LIN {X 0,Y 305.472,Z 165.433,A -85,B 0,C 180,E1 -15814.078,E2 -15814.078} C_VEL
LIN {X 0,Y 305.453,Z 165.439,A -85,B 0,C 180,E1 -15818.399,E2 -15818.399} C_VEL
LIN {X 0,Y 305.502,Z 165.428,A -85,B 0,C 180,E1 -15821.212,E2 -15821.212} C_VEL
LIN {X 0,Y 305.572,Z 165.418,A -85,B 0,C 180,E1 -15825.345,E2 -15825.345} C_VEL
LIN {X 0,Y 305.615,Z 165.414,A -85,B 0,C 180,E1 -15829.399,E2 -15829.399} C_VEL
LIN {X 0,Y 305.74,Z 165.403,A -85,B 0,C 180,E1 -15832.072,E2 -15832.072} C_VEL
LIN {X 0,Y 305.65,Z 165.409,A -85,B 0,C 180,E1 -15834.722,E2 -15834.722} C_VEL
LIN {X 0,Y 305.927,Z 165.375,A -85,B 0,C 180,E1 -15838.683,E2 -15838.683} C_VEL
LIN {X 0,Y 305.927,Z 165.375,A -85,B 0,C 180,E1 -15841.316,E2 -15841.316} C_VEL
LIN {X 0,Y 305.778,Z 165.393,A -85,B 0,C 180,E1 -15846.599,E2 -15846.599} C_VEL
LIN {X 0,Y 305.687,Z 165.406,A -85,B 0,C 180,E1 -15849.261,E2 -15849.261} C_VEL
LIN {X 0,Y 305.562,Z 165.422,A -85,B 0,C 180,E1 -15853.297,E2 -15853.297} C_VEL
LIN {X 0,Y 305.503,Z 165.429,A -85,B 0,C 180,E1 -15856.025,E2 -15856.025} C_VEL
LIN {X 0,Y 305.465,Z 165.432,A -85,B 0,C 180,E1 -15860.189,E2 -15860.189} C_VEL
LIN {X 0,Y 305.432,Z 165.436,A -85,B 0,C 180,E1 -15864.468,E2 -15864.468} C_VEL
LIN {X 0,Y 305.441,Z 165.44,A -85,B 0,C 180,E1 -15867.399,E2 -15867.399} C_VEL
LIN {X 0,Y 305.422,Z 165.437,A -85,B 0,C 180,E1 -15870.413,E2 -15870.413} C_VEL
LIN {X 0,Y 305.458,Z 165.433,A -85,B 0,C 180,E1 -15874.079,E2 -15874.079} C_VEL
LIN {X 0,Y 305.446,Z 165.435,A -85,B 0,C 180,E1 -15876.743,E2 -15876.743} C_VEL
LIN {X 0,Y 305.403,Z 165.441,A -85,B 0,C 180,E1 -15880.59,E2 -15880.59} C_VEL
LIN {X 0,Y 305.414,Z 165.439,A -85,B 0,C 180,E1 -15883.657,E2 -15883.657} C_VEL
LIN {X 0,Y 305.429,Z 165.438,A -85,B 0,C 180,E1 -15887.42,E2 -15887.42} C_VEL
LIN {X 0,Y 305.455,Z 165.434,A -85,B 0,C 180,E1 -15891.596,E2 -15891.596} C_VEL
LIN {X 0,Y 305.457,Z 165.438,A -85,B 0,C 180,E1 -15894.888,E2 -15894.888} C_VEL
LIN {X 0,Y 305.476,Z 165.491,A -85,B 0,C 180,E1 -15898.875,E2 -15898.875} C_VEL
LIN {X 0,Y 308.066,Z 178.627,A -85,B 0,C 180,E1 -15902.855,E2 -15902.855} C_VEL
LIN {X 0,Y 309.134,Z 185.066,A -85,B 0,C 180,E1 -15904.733,E2 -15904.733} C_VEL
LIN {X 0,Y 308.784,Z 188.883,A -85,B 0,C 180,E1 -15905.779,E2 -15905.779} C_VEL
LIN {X 0,Y 313.815,Z 227.795,A -85,B 0,C 180,E1 -15907.228,E2 -15907.228} C_VEL
LIN {X 0,Y 311.768,Z 298.034,A -85,B 0,C 180,E1 -15909.205,E2 -15909.205} C_VEL
LIN {X 0,Y 311.014,Z 311.572,A -85,B 0,C 180,E1 -15909.844,E2 -15909.844} C_VEL
LIN {X 0,Y 310.145,Z 323.511,A -85,B 0,C 180,E1 -15910.647,E2 -15910.647} C_VEL
LIN {X 0,Y 309.009,Z 336.037,A -85,B 0,C 180,E1 -15911.778,E2 -15911.778} C_VEL
LIN {X 0,Y 307.83,Z 347.584,A -85,B 0,C 180,E1 -15913.112,E2 -15913.112} C_VEL
LIN {X 0,Y 306.764,Z 358.549,A -85,B 0,C 180,E1 -15914.725,E2 -15914.725} C_VEL
LIN {X 0,Y 305.802,Z 367.631,A -85,B 0,C 180,E1 -15916.376,E2 -15916.376} C_VEL
LIN {X 0,Y 304.946,Z 375.108,A -85,B 0,C 180,E1 -15918.03,E2 -15918.03} C_VEL
LIN {X 0,Y 304.346,Z 382.452,A -85,B 0,C 180,E1 -15920.028,E2 -15920.028} C_VEL
LIN {X 0,Y 303.939,Z 388.258,A -85,B 0,C 180,E1 -15922.026,E2 -15922.026} C_VEL
LIN {X 0,Y 303.666,Z 393.461,A -85,B 0,C 180,E1 -15924.375,E2 -15924.375} C_VEL
LIN {X 0,Y 303.654,Z 396.168,A -85,B 0,C 180,E1 -15926.02,E2 -15926.02} C_VEL
LIN {X 0,Y 303.618,Z 397.825,A -85,B 0,C 180,E1 -15927.348,E2 -15927.348} C_VEL
LIN {X 0,Y 303.582,Z 399.055,A -85,B 0,C 180,E1 -15928.675,E2 -15928.675} C_VEL
LIN {X 0,Y 303.607,Z 399.819,A -85,B 0,C 180,E1 -15930.001,E2 -15930.001} C_VEL
LIN {X 0,Y 303.565,Z 400.151,A -85,B 0,C 180,E1 -15931.328,E2 -15931.328} C_VEL
LIN {X 0,Y 303.601,Z 400.076,A -85,B 0,C 180,E1 -15932.655,E2 -15932.655} C_VEL
LIN {X 0,Y 303.591,Z 399.592,A -85,B 0,C 180,E1 -15933.983,E2 -15933.983} C_VEL
LIN {X 0,Y 303.625,Z 398.44,A -85,B 0,C 180,E1 -15935.546,E2 -15935.546} C_VEL
LIN {X 0,Y 304.036,Z 395.535,A -85,B 0,C 180,E1 -15937.973,E2 -15937.973} C_VEL
LIN {X 0,Y 304.61,Z 392.021,A -85,B 0,C 180,E1 -15939.966,E2 -15939.966} C_VEL
LIN {X 0,Y 305.477,Z 387.416,A -85,B 0,C 180,E1 -15941.951,E2 -15941.951} C_VEL
LIN {X 0,Y 306.627,Z 381.601,A -85,B 0,C 180,E1 -15943.927,E2 -15943.927} C_VEL
LIN {X 0,Y 308.262,Z 374.337,A -85,B 0,C 180,E1 -15945.879,E2 -15945.879} C_VEL
LIN {X 0,Y 310.051,Z 365.064,A -85,B 0,C 180,E1 -15947.882,E2 -15947.882} C_VEL
LIN {X 0,Y 312.002,Z 355.271,A -85,B 0,C 180,E1 -15949.578,E2 -15949.578} C_VEL
LIN {X 0,Y 314.276,Z 343.752,A -85,B 0,C 180,E1 -15951.138,E2 -15951.138} C_VEL
LIN {X 0,Y 316.217,Z 332.295,A -85,B 0,C 180,E1 -15952.372,E2 -15952.372} C_VEL
LIN {X 0,Y 317.969,Z 319.356,A -85,B 0,C 180,E1 -15953.445,E2 -15953.445} C_VEL
LIN {X 0,Y 319.623,Z 306.314,A -85,B 0,C 180,E1 -15954.22,E2 -15954.22} C_VEL
LIN {X 0,Y 320.675,Z 292.777,A -85,B 0,C 180,E1 -15954.774,E2 -15954.774} C_VEL
LIN {X 0,Y 323.701,Z 230.457,A -85,B 0,C 180,E1 -15956.607,E2 -15956.607} C_VEL
LIN {X 0,Y 321.649,Z 216.499,A -85,B 0,C 180,E1 -15957.392,E2 -15957.392} C_VEL
LIN {X 0,Y 318.885,Z 202.613,A -85,B 0,C 180,E1 -15958.296,E2 -15958.296} C_VEL
LIN {X 0,Y 314.226,Z 192.61,A -85,B 0,C 180,E1 -15959.393,E2 -15959.393} C_VEL
LIN {X 0,Y 311.037,Z 185.839,A -85,B 0,C 180,E1 -15960.213,E2 -15960.213} C_VEL
LIN {X 0,Y 309.147,Z 178.305,A -85,B 0,C 180,E1 -15963.067,E2 -15963.067} C_VEL
LIN {X 0,Y 307.457,Z 172.034,A -85,B 0,C 180,E1 -15965.654,E2 -15965.654} C_VEL
LIN {X 0,Y 305.463,Z 165.437,A -85,B 0,C 180,E1 -15968.727,E2 -15968.727} C_VEL
LIN {X 0,Y 305.437,Z 165.436,A -85,B 0,C 180,E1 -15972.582,E2 -15972.582} C_VEL
LIN {X 0,Y 305.424,Z 165.43,A -85,B 0,C 180,E1 -15976.345,E2 -15976.345} C_VEL
LIN {X 0,Y 305.413,Z 165.437,A -85,B 0,C 180,E1 -15979.885,E2 -15979.885} C_VEL
LIN {X 0,Y 305.465,Z 165.429,A -85,B 0,C 180,E1 -15983.637,E2 -15983.637} C_VEL
LIN {X 0,Y 305.468,Z 165.43,A -85,B 0,C 180,E1 -15986.484,E2 -15986.484} C_VEL
LIN {X 0,Y 305.433,Z 165.434,A -85,B 0,C 180,E1 -15989.588,E2 -15989.588} C_VEL
LIN {X 0,Y 305.453,Z 165.433,A -85,B 0,C 180,E1 -15992.602,E2 -15992.602} C_VEL
LIN {X 0,Y 305.459,Z 165.434,A -85,B 0,C 180,E1 -15995.535,E2 -15995.535} C_VEL
LIN {X 0,Y 305.483,Z 165.428,A -85,B 0,C 180,E1 -15999.813,E2 -15999.813} C_VEL
LIN {X 0,Y 305.518,Z 165.426,A -85,B 0,C 180,E1 -16003.976,E2 -16003.976} C_VEL
LIN {X 0,Y 305.576,Z 165.421,A -85,B 0,C 180,E1 -16006.704,E2 -16006.704} C_VEL
LIN {X 0,Y 305.758,Z 165.403,A -85,B 0,C 180,E1 -16011.262,E2 -16011.262} C_VEL
LIN {X 0,Y 305.814,Z 165.503,A -85,B 0,C 180,E1 -16013.319,E2 -16013.319} C_VEL
LIN {X 0,Y 308.783,Z 174.874,A -85,B 0,C 180,E1 -16017.493,E2 -16017.493} C_VEL
LIN {X 0,Y 316.098,Z 187.842,A -85,B 0,C 180,E1 -16019.227,E2 -16019.227} C_VEL
LIN {X 0,Y 320.795,Z 197.781,A -85,B 0,C 180,E1 -16020.318,E2 -16020.318} C_VEL
LIN {X 0,Y 324.339,Z 206.07,A -85,B 0,C 180,E1 -16021.105,E2 -16021.105} C_VEL
LIN {X 0,Y 324.803,Z 209.109,A -85,B 0,C 180,E1 -16021.277,E2 -16021.277} C_VEL
LIN {X 0,Y 320.791,Z 283.034,A -85,B 0,C 180,E1 -16023.454,E2 -16023.454} C_VEL
LIN {X 0,Y 319.653,Z 296.49,A -85,B 0,C 180,E1 -16024.098,E2 -16024.098} C_VEL
LIN {X 0,Y 318.359,Z 308.395,A -85,B 0,C 180,E1 -16024.908,E2 -16024.908} C_VEL
LIN {X 0,Y 316.679,Z 320.8,A -85,B 0,C 180,E1 -16026.033,E2 -16026.033} C_VEL
LIN {X 0,Y 314.754,Z 332.399,A -85,B 0,C 180,E1 -16027.377,E2 -16027.377} C_VEL
LIN {X 0,Y 312.921,Z 342.14,A -85,B 0,C 180,E1 -16028.802,E2 -16028.802} C_VEL
LIN {X 0,Y 311.039,Z 351.123,A -85,B 0,C 180,E1 -16030.415,E2 -16030.415} C_VEL
LIN {X 0,Y 309.272,Z 359.452,A -85,B 0,C 180,E1 -16032.269,E2 -16032.269} C_VEL
LIN {X 0,Y 307.722,Z 366.472,A -85,B 0,C 180,E1 -16034.213,E2 -16034.213} C_VEL
LIN {X 0,Y 306.509,Z 371.582,A -85,B 0,C 180,E1 -16035.971,E2 -16035.971} C_VEL
LIN {X 0,Y 305.397,Z 376.396,A -85,B 0,C 180,E1 -16038.1,E2 -16038.1} C_VEL
LIN {X 0,Y 304.623,Z 379.954,A -85,B 0,C 180,E1 -16040.247,E2 -16040.247} C_VEL
LIN {X 0,Y 304.009,Z 382.327,A -85,B 0,C 180,E1 -16042.373,E2 -16042.373} C_VEL
LIN {X 0,Y 303.584,Z 383.655,A -85,B 0,C 180,E1 -16044.627,E2 -16044.627} C_VEL
LIN {X 0,Y 303.405,Z 383.901,A -85,B 0,C 180,E1 -16046.112,E2 -16046.112} C_VEL
LIN {X 0,Y 303.329,Z 383.27,A -85,B 0,C 180,E1 -16048.302,E2 -16048.302} C_VEL
LIN {X 0,Y 303.429,Z 380.868,A -85,B 0,C 180,E1 -16051.018,E2 -16051.018} C_VEL
LIN {X 0,Y 303.701,Z 378.144,A -85,B 0,C 180,E1 -16052.891,E2 -16052.891} C_VEL
LIN {X 0,Y 304.053,Z 373.262,A -85,B 0,C 180,E1 -16055.301,E2 -16055.301} C_VEL
LIN {X 0,Y 304.626,Z 366.761,A -85,B 0,C 180,E1 -16057.64,E2 -16057.64} C_VEL
LIN {X 0,Y 305.372,Z 359.46,A -85,B 0,C 180,E1 -16059.692,E2 -16059.692} C_VEL
LIN {X 0,Y 306.156,Z 351.81,A -85,B 0,C 180,E1 -16061.427,E2 -16061.427} C_VEL
LIN {X 0,Y 307.049,Z 342.979,A -85,B 0,C 180,E1 -16063.065,E2 -16063.065} C_VEL
LIN {X 0,Y 308.206,Z 331.704,A -85,B 0,C 180,E1 -16064.753,E2 -16064.753} C_VEL
LIN {X 0,Y 309.372,Z 319.69,A -85,B 0,C 180,E1 -16066.164,E2 -16066.164} C_VEL
LIN {X 0,Y 310.388,Z 307.413,A -85,B 0,C 180,E1 -16067.287,E2 -16067.287} C_VEL
LIN {X 0,Y 311.251,Z 294.444,A -85,B 0,C 180,E1 -16068.172,E2 -16068.172} C_VEL
LIN {X 0,Y 311.848,Z 281.457,A -85,B 0,C 180,E1 -16068.79,E2 -16068.79} C_VEL
LIN {X 0,Y 313.435,Z 231.762,A -85,B 0,C 180,E1 -16070.193,E2 -16070.193} C_VEL
LIN {X 0,Y 314.134,Z 202.407,A -85,B 0,C 180,E1 -16071.018,E2 -16071.018} C_VEL
LIN {X 0,Y 311.365,Z 186.836,A -85,B 0,C 180,E1 -16071.635,E2 -16071.635} C_VEL
LIN {X 0,Y 306.865,Z 172.397,A -85,B 0,C 180,E1 -16072.373,E2 -16072.373} C_VEL
LIN {X 0,Y 305.523,Z 165.429,A -85,B 0,C 180,E1 -16074.692,E2 -16074.692} C_VEL
LIN {X 0,Y 305.447,Z 165.439,A -85,B 0,C 180,E1 -16078.358,E2 -16078.358} C_VEL
LIN {X 0,Y 305.458,Z 165.434,A -85,B 0,C 180,E1 -16081.106,E2 -16081.106} C_VEL
LIN {X 0,Y 305.483,Z 165.433,A -85,B 0,C 180,E1 -16084.079,E2 -16084.079} C_VEL
LIN {X 0,Y 305.463,Z 165.436,A -85,B 0,C 180,E1 -16088.399,E2 -16088.399} C_VEL
LIN {X 0,Y 305.506,Z 165.427,A -85,B 0,C 180,E1 -16091.211,E2 -16091.211} C_VEL
LIN {X 0,Y 305.583,Z 165.418,A -85,B 0,C 180,E1 -16095.345,E2 -16095.345} C_VEL
LIN {X 0,Y 305.627,Z 165.413,A -85,B 0,C 180,E1 -16099.398,E2 -16099.398} C_VEL
LIN {X 0,Y 305.751,Z 165.401,A -85,B 0,C 180,E1 -16102.072,E2 -16102.072} C_VEL
LIN {X 0,Y 305.66,Z 165.408,A -85,B 0,C 180,E1 -16104.722,E2 -16104.722} C_VEL
LIN {X 0,Y 305.939,Z 165.373,A -85,B 0,C 180,E1 -16108.683,E2 -16108.683} C_VEL
LIN {X 0,Y 305.939,Z 165.374,A -85,B 0,C 180,E1 -16111.315,E2 -16111.315} C_VEL
LIN {X 0,Y 305.787,Z 165.392,A -85,B 0,C 180,E1 -16116.598,E2 -16116.598} C_VEL
LIN {X 0,Y 305.697,Z 165.405,A -85,B 0,C 180,E1 -16119.26,E2 -16119.26} C_VEL
LIN {X 0,Y 305.572,Z 165.422,A -85,B 0,C 180,E1 -16123.296,E2 -16123.296} C_VEL
LIN {X 0,Y 305.512,Z 165.427,A -85,B 0,C 180,E1 -16126.023,E2 -16126.023} C_VEL
LIN {X 0,Y 305.473,Z 165.431,A -85,B 0,C 180,E1 -16130.187,E2 -16130.187} C_VEL
LIN {X 0,Y 305.44,Z 165.435,A -85,B 0,C 180,E1 -16134.466,E2 -16134.466} C_VEL
LIN {X 0,Y 305.449,Z 165.438,A -85,B 0,C 180,E1 -16137.397,E2 -16137.397} C_VEL
LIN {X 0,Y 305.428,Z 165.437,A -85,B 0,C 180,E1 -16140.411,E2 -16140.411} C_VEL
LIN {X 0,Y 305.463,Z 165.432,A -85,B 0,C 180,E1 -16144.077,E2 -16144.077} C_VEL
LIN {X 0,Y 305.451,Z 165.436,A -85,B 0,C 180,E1 -16146.741,E2 -16146.741} C_VEL
LIN {X 0,Y 305.407,Z 165.441,A -85,B 0,C 180,E1 -16150.588,E2 -16150.588} C_VEL
LIN {X 0,Y 305.418,Z 165.438,A -85,B 0,C 180,E1 -16153.655,E2 -16153.655} C_VEL
LIN {X 0,Y 305.431,Z 165.437,A -85,B 0,C 180,E1 -16157.417,E2 -16157.417} C_VEL
LIN {X 0,Y 305.456,Z 165.433,A -85,B 0,C 180,E1 -16161.594,E2 -16161.594} C_VEL
LIN {X 0,Y 305.441,Z 165.435,A -85,B 0,C 180,E1 -16164.445,E2 -16164.445} C_VEL
LIN {X 0,Y 304.777,Z 165.521,A -85,B 0,C 180,E1 -16165.546,E2 -16165.546} C_VEL
LIN {X 0,Y 301.877,Z 165.879,A -85,B 0,C 180,E1 -16167.337,E2 -16167.337} C_VEL
LIN {X 0,Y 299.44,Z 166.186,A -85,B 0,C 180,E1 -16168.791,E2 -16168.791} C_VEL
LIN {X 0,Y 298.44,Z 166.308,A -85,B 0,C 180,E1 -16169.918,E2 -16169.918} C_VEL
LIN {X 0,Y 298.383,Z 166.317,A -85,B 0,C 180,E1 -16170.299,E2 -16170.299} C_VEL
LIN {X 0,Y 298.398,Z 166.312,A -85,B 0,C 180,E1 -16173.504,E2 -16173.504} C_VEL
LIN {X 0,Y 298.399,Z 166.314,A -85,B 0,C 180,E1 -16176.71,E2 -16176.71} C_VEL
LIN {X 0,Y 298.453,Z 166.307,A -85,B 0,C 180,E1 -16180.751,E2 -16180.751} C_VEL
LIN {X 0,Y 298.504,Z 166.299,A -85,B 0,C 180,E1 -16184.99,E2 -16184.99} C_VEL
LIN {X 0,Y 298.574,Z 166.291,A -85,B 0,C 180,E1 -16189.146,E2 -16189.146} C_VEL
LIN {X 0,Y 298.691,Z 166.279,A -85,B 0,C 180,E1 -16191.884,E2 -16191.884} C_VEL
LIN {X 0,Y 298.62,Z 166.285,A -85,B 0,C 180,E1 -16194.598,E2 -16194.598} C_VEL
LIN {X 0,Y 298.895,Z 166.251,A -85,B 0,C 180,E1 -16198.652,E2 -16198.652} C_VEL
LIN {X 0,Y 298.895,Z 166.251,A -85,B 0,C 180,E1 -16201.347,E2 -16201.347} C_VEL
LIN {X 0,Y 298.727,Z 166.271,A -85,B 0,C 180,E1 -16206.755,E2 -16206.755} C_VEL
LIN {X 0,Y 298.618,Z 166.288,A -85,B 0,C 180,E1 -16209.482,E2 -16209.482} C_VEL
LIN {X 0,Y 298.515,Z 166.303,A -85,B 0,C 180,E1 -16213.617,E2 -16213.617} C_VEL
LIN {X 0,Y 298.443,Z 166.307,A -85,B 0,C 180,E1 -16216.414,E2 -16216.414} C_VEL
LIN {X 0,Y 298.422,Z 166.314,A -85,B 0,C 180,E1 -16219.61,E2 -16219.61} C_VEL
LIN {X 0,Y 298.375,Z 166.319,A -85,B 0,C 180,E1 -16223.604,E2 -16223.604} C_VEL
LIN {X 0,Y 298.395,Z 166.313,A -85,B 0,C 180,E1 -16226.583,E2 -16226.583} C_VEL
LIN {X 0,Y 298.385,Z 166.316,A -85,B 0,C 180,E1 -16229.645,E2 -16229.645} C_VEL
LIN {X 0,Y 298.386,Z 166.315,A -85,B 0,C 180,E1 -16232.801,E2 -16232.801} C_VEL
LIN {X 0,Y 298.421,Z 166.311,A -85,B 0,C 180,E1 -16236.803,E2 -16236.803} C_VEL
LIN {X 0,Y 298.367,Z 166.318,A -85,B 0,C 180,E1 -16239.493,E2 -16239.493} C_VEL
LIN {X 0,Y 298.364,Z 166.322,A -85,B 0,C 180,E1 -16243.098,E2 -16243.098} C_VEL
LIN {X 0,Y 298.365,Z 166.322,A -85,B 0,C 180,E1 -16246.916,E2 -16246.916} C_VEL
LIN {X 0,Y 298.379,Z 166.319,A -85,B 0,C 180,E1 -16251.012,E2 -16251.012} C_VEL
LIN {X 0,Y 298.4,Z 166.312,A -85,B 0,C 180,E1 -16253.929,E2 -16253.929} C_VEL
LIN {X 0,Y 298.389,Z 166.317,A -85,B 0,C 180,E1 -16257.201,E2 -16257.201} C_VEL
LIN {X 0,Y 298.415,Z 166.357,A -85,B 0,C 180,E1 -16258.581,E2 -16258.581} C_VEL
LIN {X 0,Y 300.976,Z 179.093,A -85,B 0,C 180,E1 -16262.539,E2 -16262.539} C_VEL
LIN {X 0,Y 302.103,Z 185.693,A -85,B 0,C 180,E1 -16264.511,E2 -16264.511} C_VEL
LIN {X 0,Y 301.911,Z 188.736,A -85,B 0,C 180,E1 -16265.371,E2 -16265.371} C_VEL
LIN {X 0,Y 306.968,Z 229.189,A -85,B 0,C 180,E1 -16266.912,E2 -16266.912} C_VEL
LIN {X 0,Y 304.887,Z 297.637,A -85,B 0,C 180,E1 -16268.89,E2 -16268.89} C_VEL
LIN {X 0,Y 304.135,Z 311.222,A -85,B 0,C 180,E1 -16269.544,E2 -16269.544} C_VEL
LIN {X 0,Y 303.23,Z 323.192,A -85,B 0,C 180,E1 -16270.364,E2 -16270.364} C_VEL
LIN {X 0,Y 302.05,Z 335.742,A -85,B 0,C 180,E1 -16271.518,E2 -16271.518} C_VEL
LIN {X 0,Y 300.83,Z 347.439,A -85,B 0,C 180,E1 -16272.9,E2 -16272.9} C_VEL
LIN {X 0,Y 299.791,Z 357.614,A -85,B 0,C 180,E1 -16274.417,E2 -16274.417} C_VEL
LIN {X 0,Y 298.817,Z 366.553,A -85,B 0,C 180,E1 -16276.051,E2 -16276.051} C_VEL
LIN {X 0,Y 297.828,Z 375.581,A -85,B 0,C 180,E1 -16278.085,E2 -16278.085} C_VEL
LIN {X 0,Y 297.207,Z 382.758,A -85,B 0,C 180,E1 -16280.13,E2 -16280.13} C_VEL
LIN {X 0,Y 296.785,Z 389.304,A -85,B 0,C 180,E1 -16282.518,E2 -16282.518} C_VEL
LIN {X 0,Y 296.58,Z 393.545,A -85,B 0,C 180,E1 -16284.562,E2 -16284.562} C_VEL
LIN {X 0,Y 296.566,Z 395.739,A -85,B 0,C 180,E1 -16285.924,E2 -16285.924} C_VEL
LIN {X 0,Y 296.545,Z 397.441,A -85,B 0,C 180,E1 -16287.284,E2 -16287.284} C_VEL
LIN {X 0,Y 296.501,Z 398.713,A -85,B 0,C 180,E1 -16288.643,E2 -16288.643} C_VEL
LIN {X 0,Y 296.521,Z 399.555,A -85,B 0,C 180,E1 -16290.001,E2 -16290.001} C_VEL
LIN {X 0,Y 296.485,Z 399.929,A -85,B 0,C 180,E1 -16291.359,E2 -16291.359} C_VEL
LIN {X 0,Y 296.525,Z 399.894,A -85,B 0,C 180,E1 -16292.718,E2 -16292.718} C_VEL
LIN {X 0,Y 296.491,Z 399.454,A -85,B 0,C 180,E1 -16294.079,E2 -16294.079} C_VEL
LIN {X 0,Y 296.546,Z 398.537,A -85,B 0,C 180,E1 -16295.51,E2 -16295.51} C_VEL
LIN {X 0,Y 296.986,Z 395.571,A -85,B 0,C 180,E1 -16298.164,E2 -16298.164} C_VEL
LIN {X 0,Y 297.591,Z 392.145,A -85,B 0,C 180,E1 -16300.203,E2 -16300.203} C_VEL
LIN {X 0,Y 298.507,Z 387.63,A -85,B 0,C 180,E1 -16302.235,E2 -16302.235} C_VEL
LIN {X 0,Y 299.758,Z 381.92,A -85,B 0,C 180,E1 -16304.253,E2 -16304.253} C_VEL
LIN {X 0,Y 301.466,Z 374.857,A -85,B 0,C 180,E1 -16306.247,E2 -16306.247} C_VEL
LIN {X 0,Y 303.31,Z 365.962,A -85,B 0,C 180,E1 -16308.257,E2 -16308.257} C_VEL
LIN {X 0,Y 305.241,Z 357.152,A -85,B 0,C 180,E1 -16309.854,E2 -16309.854} C_VEL
LIN {X 0,Y 307.472,Z 346.24,A -85,B 0,C 180,E1 -16311.453,E2 -16311.453} C_VEL
LIN {X 0,Y 309.771,Z 333.801,A -85,B 0,C 180,E1 -16312.864,E2 -16312.864} C_VEL
LIN {X 0,Y 311.583,Z 321.633,A -85,B 0,C 180,E1 -16313.955,E2 -16313.955} C_VEL
LIN {X 0,Y 313.417,Z 308.119,A -85,B 0,C 180,E1 -16314.82,E2 -16314.82} C_VEL
LIN {X 0,Y 314.688,Z 294.787,A -85,B 0,C 180,E1 -16315.419,E2 -16315.419} C_VEL
LIN {X 0,Y 317.963,Z 231.766,A -85,B 0,C 180,E1 -16317.319,E2 -16317.319} C_VEL
LIN {X 0,Y 315.972,Z 217.769,A -85,B 0,C 180,E1 -16318.133,E2 -16318.133} C_VEL
LIN {X 0,Y 313.691,Z 206.025,A -85,B 0,C 180,E1 -16318.94,E2 -16318.94} C_VEL
LIN {X 0,Y 308.299,Z 194.321,A -85,B 0,C 180,E1 -16320.281,E2 -16320.281} C_VEL
LIN {X 0,Y 305.45,Z 188.925,A -85,B 0,C 180,E1 -16321.007,E2 -16321.007} C_VEL
LIN {X 0,Y 303.831,Z 185.519,A -85,B 0,C 180,E1 -16321.484,E2 -16321.484} C_VEL
LIN {X 0,Y 301.449,Z 176.169,A -85,B 0,C 180,E1 -16325.314,E2 -16325.314} C_VEL
LIN {X 0,Y 299.296,Z 169.326,A -85,B 0,C 180,E1 -16328.55,E2 -16328.55} C_VEL
LIN {X 0,Y 298.379,Z 166.317,A -85,B 0,C 180,E1 -16330.151,E2 -16330.151} C_VEL
LIN {X 0,Y 298.373,Z 166.315,A -85,B 0,C 180,E1 -16333.098,E2 -16333.098} C_VEL
LIN {X 0,Y 298.373,Z 166.309,A -85,B 0,C 180,E1 -16336.916,E2 -16336.916} C_VEL
LIN {X 0,Y 298.388,Z 166.308,A -85,B 0,C 180,E1 -16341.012,E2 -16341.012} C_VEL
LIN {X 0,Y 298.407,Z 166.308,A -85,B 0,C 180,E1 -16343.929,E2 -16343.929} C_VEL
LIN {X 0,Y 298.396,Z 166.313,A -85,B 0,C 180,E1 -16347.2,E2 -16347.2} C_VEL
LIN {X 0,Y 298.405,Z 166.314,A -85,B 0,C 180,E1 -16350.626,E2 -16350.626} C_VEL
LIN {X 0,Y 298.425,Z 166.307,A -85,B 0,C 180,E1 -16354.919,E2 -16354.919} C_VEL
LIN {X 0,Y 298.419,Z 166.306,A -85,B 0,C 180,E1 -16359.313,E2 -16359.313} C_VEL
LIN {X 0,Y 298.452,Z 166.306,A -85,B 0,C 180,E1 -16362.174,E2 -16362.174} C_VEL
LIN {X 0,Y 298.515,Z 166.303,A -85,B 0,C 180,E1 -16364.991,E2 -16364.991} C_VEL
LIN {X 0,Y 298.587,Z 166.296,A -85,B 0,C 180,E1 -16369.147,E2 -16369.147} C_VEL
LIN {X 0,Y 298.713,Z 166.37,A -85,B 0,C 180,E1 -16371.885,E2 -16371.885} C_VEL
LIN {X 0,Y 299.956,Z 170.371,A -85,B 0,C 180,E1 -16373.948,E2 -16373.948} C_VEL
LIN {X 0,Y 301.337,Z 175.242,A -85,B 0,C 180,E1 -16376.139,E2 -16376.139} C_VEL
LIN {X 0,Y 304.291,Z 179.547,A -85,B 0,C 180,E1 -16376.897,E2 -16376.897} C_VEL
LIN {X 0,Y 311.305,Z 192.016,A -85,B 0,C 180,E1 -16378.646,E2 -16378.646} C_VEL
LIN {X 0,Y 316.01,Z 202.117,A -85,B 0,C 180,E1 -16379.779,E2 -16379.779} C_VEL
LIN {X 0,Y 318.965,Z 209.24,A -85,B 0,C 180,E1 -16380.494,E2 -16380.494} C_VEL
LIN {X 0,Y 318.072,Z 227.571,A -85,B 0,C 180,E1 -16381.061,E2 -16381.061} C_VEL
LIN {X 0,Y 314.991,Z 282.686,A -85,B 0,C 180,E1 -16382.718,E2 -16382.718} C_VEL
LIN {X 0,Y 313.782,Z 296.248,A -85,B 0,C 180,E1 -16383.371,E2 -16383.371} C_VEL
LIN {X 0,Y 312.23,Z 309.274,A -85,B 0,C 180,E1 -16384.276,E2 -16384.276} C_VEL
LIN {X 0,Y 310.419,Z 321.832,A -85,B 0,C 180,E1 -16385.46,E2 -16385.46} C_VEL
LIN {X 0,Y 308.303,Z 333.575,A -85,B 0,C 180,E1 -16386.874,E2 -16386.874} C_VEL
LIN {X 0,Y 306.059,Z 344.76,A -85,B 0,C 180,E1 -16388.592,E2 -16388.592} C_VEL
LIN {X 0,Y 304.069,Z 353.697,A -85,B 0,C 180,E1 -16390.319,E2 -16390.319} C_VEL
LIN {X 0,Y 302.142,Z 361.956,A -85,B 0,C 180,E1 -16392.323,E2 -16392.323} C_VEL
LIN {X 0,Y 300.35,Z 369.263,A -85,B 0,C 180,E1 -16394.569,E2 -16394.569} C_VEL
LIN {X 0,Y 298.812,Z 375.42,A -85,B 0,C 180,E1 -16397.098,E2 -16397.098} C_VEL
LIN {X 0,Y 297.873,Z 379.354,A -85,B 0,C 180,E1 -16399.305,E2 -16399.305} C_VEL
LIN {X 0,Y 297.361,Z 381.278,A -85,B 0,C 180,E1 -16400.764,E2 -16400.764} C_VEL
LIN {X 0,Y 296.879,Z 382.975,A -85,B 0,C 180,E1 -16402.592,E2 -16402.592} C_VEL
LIN {X 0,Y 296.632,Z 383.657,A -85,B 0,C 180,E1 -16403.752,E2 -16403.752} C_VEL
LIN {X 0,Y 296.374,Z 384.096,A -85,B 0,C 180,E1 -16405.694,E2 -16405.694} C_VEL
LIN {X 0,Y 296.238,Z 383.358,A -85,B 0,C 180,E1 -16408.326,E2 -16408.326} C_VEL
LIN {X 0,Y 296.262,Z 382.178,A -85,B 0,C 180,E1 -16409.879,E2 -16409.879} C_VEL
LIN {X 0,Y 296.51,Z 379.335,A -85,B 0,C 180,E1 -16412.23,E2 -16412.23} C_VEL
LIN {X 0,Y 296.872,Z 374.965,A -85,B 0,C 180,E1 -16414.623,E2 -16414.623} C_VEL
LIN {X 0,Y 297.194,Z 370.485,A -85,B 0,C 180,E1 -16416.482,E2 -16416.482} C_VEL
LIN {X 0,Y 297.764,Z 364.753,A -85,B 0,C 180,E1 -16418.384,E2 -16418.384} C_VEL
LIN {X 0,Y 298.532,Z 357.413,A -85,B 0,C 180,E1 -16420.347,E2 -16420.347} C_VEL
LIN {X 0,Y 299.483,Z 348.857,A -85,B 0,C 180,E1 -16422.202,E2 -16422.202} C_VEL
LIN {X 0,Y 300.445,Z 339.005,A -85,B 0,C 180,E1 -16423.93,E2 -16423.93} C_VEL
LIN {X 0,Y 301.689,Z 327.13,A -85,B 0,C 180,E1 -16425.586,E2 -16425.586} C_VEL
LIN {X 0,Y 302.812,Z 315.497,A -85,B 0,C 180,E1 -16426.857,E2 -16426.857} C_VEL
LIN {X 0,Y 303.814,Z 302.479,A -85,B 0,C 180,E1 -16427.953,E2 -16427.953} C_VEL
LIN {X 0,Y 304.554,Z 289.194,A -85,B 0,C 180,E1 -16428.765,E2 -16428.765} C_VEL
LIN {X 0,Y 305.233,Z 275.398,A -85,B 0,C 180,E1 -16429.31,E2 -16429.31} C_VEL
LIN {X 0,Y 307.384,Z 203.753,A -85,B 0,C 180,E1 -16431.347,E2 -16431.347} C_VEL
LIN {X 0,Y 304.735,Z 188.686,A -85,B 0,C 180,E1 -16431.96,E2 -16431.96} C_VEL
LIN {X 0,Y 299.72,Z 172.714,A -85,B 0,C 180,E1 -16432.77,E2 -16432.77} C_VEL
LIN {X 0,Y 298.492,Z 166.303,A -85,B 0,C 180,E1 -16434.925,E2 -16434.925} C_VEL
LIN {X 0,Y 298.377,Z 166.318,A -85,B 0,C 180,E1 -16438.788,E2 -16438.788} C_VEL
LIN {X 0,Y 298.4,Z 166.314,A -85,B 0,C 180,E1 -16441.897,E2 -16441.897} C_VEL
LIN {X 0,Y 298.417,Z 166.311,A -85,B 0,C 180,E1 -16444.917,E2 -16444.917} C_VEL
LIN {X 0,Y 298.395,Z 166.315,A -85,B 0,C 180,E1 -16447.861,E2 -16447.861} C_VEL
LIN {X 0,Y 298.457,Z 166.306,A -85,B 0,C 180,E1 -16450.75,E2 -16450.75} C_VEL
LIN {X 0,Y 298.515,Z 166.298,A -85,B 0,C 180,E1 -16454.99,E2 -16454.99} C_VEL
LIN {X 0,Y 298.586,Z 166.289,A -85,B 0,C 180,E1 -16459.145,E2 -16459.145} C_VEL
LIN {X 0,Y 298.702,Z 166.279,A -85,B 0,C 180,E1 -16461.883,E2 -16461.883} C_VEL
LIN {X 0,Y 298.63,Z 166.284,A -85,B 0,C 180,E1 -16464.597,E2 -16464.597} C_VEL
LIN {X 0,Y 298.907,Z 166.249,A -85,B 0,C 180,E1 -16468.652,E2 -16468.652} C_VEL
LIN {X 0,Y 298.906,Z 166.25,A -85,B 0,C 180,E1 -16471.346,E2 -16471.346} C_VEL
LIN {X 0,Y 298.736,Z 166.27,A -85,B 0,C 180,E1 -16476.754,E2 -16476.754} C_VEL
LIN {X 0,Y 298.628,Z 166.287,A -85,B 0,C 180,E1 -16479.481,E2 -16479.481} C_VEL
LIN {X 0,Y 298.525,Z 166.301,A -85,B 0,C 180,E1 -16483.615,E2 -16483.615} C_VEL
LIN {X 0,Y 298.452,Z 166.305,A -85,B 0,C 180,E1 -16486.413,E2 -16486.413} C_VEL
LIN {X 0,Y 298.43,Z 166.312,A -85,B 0,C 180,E1 -16489.609,E2 -16489.609} C_VEL
LIN {X 0,Y 298.382,Z 166.317,A -85,B 0,C 180,E1 -16493.603,E2 -16493.603} C_VEL
LIN {X 0,Y 298.402,Z 166.312,A -85,B 0,C 180,E1 -16496.581,E2 -16496.581} C_VEL
LIN {X 0,Y 298.392,Z 166.315,A -85,B 0,C 180,E1 -16499.643,E2 -16499.643} C_VEL
LIN {X 0,Y 298.392,Z 166.315,A -85,B 0,C 180,E1 -16502.799,E2 -16502.799} C_VEL
LIN {X 0,Y 298.425,Z 166.312,A -85,B 0,C 180,E1 -16506.801,E2 -16506.801} C_VEL
LIN {X 0,Y 298.371,Z 166.317,A -85,B 0,C 180,E1 -16509.49,E2 -16509.49} C_VEL
LIN {X 0,Y 298.368,Z 166.32,A -85,B 0,C 180,E1 -16513.096,E2 -16513.096} C_VEL
LIN {X 0,Y 298.367,Z 166.321,A -85,B 0,C 180,E1 -16516.914,E2 -16516.914} C_VEL
LIN {X 0,Y 298.38,Z 166.317,A -85,B 0,C 180,E1 -16521.01,E2 -16521.01} C_VEL
LIN {X 0,Y 298.383,Z 166.311,A -85,B 0,C 180,E1 -16524.443,E2 -16524.443} C_VEL
LIN {X 0,Y 298.383,Z 166.315,A -85,B 0,C 180,E1 -16527.985,E2 -16527.985} C_VEL
LIN {X 0,Y 298.383,Z 166.317,A -85,B 0,C 180,E1 -16530.299,E2 -16530.299} C_VEL
LIN {X 0,Y 297.766,Z 166.399,A -85,B 0,C 180,E1 -16531.427,E2 -16531.427} C_VEL
LIN {X 0,Y 294.881,Z 166.754,A -85,B 0,C 180,E1 -16533.261,E2 -16533.261} C_VEL
LIN {X 0,Y 292.422,Z 167.059,A -85,B 0,C 180,E1 -16534.75,E2 -16534.75} C_VEL
LIN {X 0,Y 291.401,Z 167.185,A -85,B 0,C 180,E1 -16535.905,E2 -16535.905} C_VEL
LIN {X 0,Y 291.339,Z 167.195,A -85,B 0,C 180,E1 -16536.296,E2 -16536.296} C_VEL
LIN {X 0,Y 291.379,Z 167.191,A -85,B 0,C 180,E1 -16540.264,E2 -16540.264} C_VEL
LIN {X 0,Y 291.467,Z 167.177,A -85,B 0,C 180,E1 -16544.682,E2 -16544.682} C_VEL
LIN {X 0,Y 291.519,Z 167.17,A -85,B 0,C 180,E1 -16548.88,E2 -16548.88} C_VEL
LIN {X 0,Y 291.645,Z 167.155,A -85,B 0,C 180,E1 -16551.686,E2 -16551.686} C_VEL
LIN {X 0,Y 291.59,Z 167.162,A -85,B 0,C 180,E1 -16554.467,E2 -16554.467} C_VEL
LIN {X 0,Y 291.863,Z 167.127,A -85,B 0,C 180,E1 -16558.62,E2 -16558.62} C_VEL
LIN {X 0,Y 291.863,Z 167.127,A -85,B 0,C 180,E1 -16561.379,E2 -16561.379} C_VEL
LIN {X 0,Y 291.679,Z 167.15,A -85,B 0,C 180,E1 -16566.919,E2 -16566.919} C_VEL
LIN {X 0,Y 291.56,Z 167.169,A -85,B 0,C 180,E1 -16569.714,E2 -16569.714} C_VEL
LIN {X 0,Y 291.473,Z 167.178,A -85,B 0,C 180,E1 -16573.952,E2 -16573.952} C_VEL
LIN {X 0,Y 291.394,Z 167.185,A -85,B 0,C 180,E1 -16576.823,E2 -16576.823} C_VEL
LIN {X 0,Y 291.384,Z 167.188,A -85,B 0,C 180,E1 -16579.842,E2 -16579.842} C_VEL
LIN {X 0,Y 291.318,Z 167.195,A -85,B 0,C 180,E1 -16584.212,E2 -16584.212} C_VEL
LIN {X 0,Y 291.342,Z 167.195,A -85,B 0,C 180,E1 -16587.279,E2 -16587.279} C_VEL
LIN {X 0,Y 291.311,Z 167.195,A -85,B 0,C 180,E1 -16590.44,E2 -16590.44} C_VEL
LIN {X 0,Y 291.337,Z 167.193,A -85,B 0,C 180,E1 -16593.699,E2 -16593.699} C_VEL
LIN {X 0,Y 291.352,Z 167.194,A -85,B 0,C 180,E1 -16597.25,E2 -16597.25} C_VEL
LIN {X 0,Y 291.294,Z 167.199,A -85,B 0,C 180,E1 -16600.649,E2 -16600.649} C_VEL
LIN {X 0,Y 291.275,Z 167.201,A -85,B 0,C 180,E1 -16604.405,E2 -16604.405} C_VEL
LIN {X 0,Y 291.289,Z 167.199,A -85,B 0,C 180,E1 -16608.412,E2 -16608.412} C_VEL
LIN {X 0,Y 291.329,Z 167.196,A -85,B 0,C 180,E1 -16611.156,E2 -16611.156} C_VEL
LIN {X 0,Y 291.35,Z 167.194,A -85,B 0,C 180,E1 -16614.626,E2 -16614.626} C_VEL
LIN {X 0,Y 291.384,Z 167.302,A -85,B 0,C 180,E1 -16618.31,E2 -16618.31} C_VEL
LIN {X 0,Y 294.096,Z 180.909,A -85,B 0,C 180,E1 -16622.632,E2 -16622.632} C_VEL
LIN {X 0,Y 295.1,Z 187.432,A -85,B 0,C 180,E1 -16624.617,E2 -16624.617} C_VEL
LIN {X 0,Y 295.003,Z 188.589,A -85,B 0,C 180,E1 -16624.951,E2 -16624.951} C_VEL
LIN {X 0,Y 300.119,Z 230.027,A -85,B 0,C 180,E1 -16626.568,E2 -16626.568} C_VEL
LIN {X 0,Y 298.017,Z 297.241,A -85,B 0,C 180,E1 -16628.561,E2 -16628.561} C_VEL
LIN {X 0,Y 297.259,Z 310.868,A -85,B 0,C 180,E1 -16629.23,E2 -16629.23} C_VEL
LIN {X 0,Y 296.32,Z 322.871,A -85,B 0,C 180,E1 -16630.067,E2 -16630.067} C_VEL
LIN {X 0,Y 295.102,Z 335.448,A -85,B 0,C 180,E1 -16631.247,E2 -16631.247} C_VEL
LIN {X 0,Y 293.906,Z 346.778,A -85,B 0,C 180,E1 -16632.609,E2 -16632.609} C_VEL
LIN {X 0,Y 292.8,Z 356.927,A -85,B 0,C 180,E1 -16634.137,E2 -16634.137} C_VEL
LIN {X 0,Y 291.846,Z 365.476,A -85,B 0,C 180,E1 -16635.711,E2 -16635.711} C_VEL
LIN {X 0,Y 291,Z 373.266,A -85,B 0,C 180,E1 -16637.447,E2 -16637.447} C_VEL
LIN {X 0,Y 290.293,Z 380.893,A -85,B 0,C 180,E1 -16639.54,E2 -16639.54} C_VEL
LIN {X 0,Y 289.828,Z 386.982,A -85,B 0,C 180,E1 -16641.635,E2 -16641.635} C_VEL
LIN {X 0,Y 289.561,Z 391.731,A -85,B 0,C 180,E1 -16643.731,E2 -16643.731} C_VEL
LIN {X 0,Y 289.465,Z 395.293,A -85,B 0,C 180,E1 -16645.824,E2 -16645.824} C_VEL
LIN {X 0,Y 289.473,Z 397.046,A -85,B 0,C 180,E1 -16647.218,E2 -16647.218} C_VEL
LIN {X 0,Y 289.422,Z 398.358,A -85,B 0,C 180,E1 -16648.61,E2 -16648.61} C_VEL
LIN {X 0,Y 289.438,Z 399.254,A -85,B 0,C 180,E1 -16650.001,E2 -16650.001} C_VEL
LIN {X 0,Y 289.406,Z 399.703,A -85,B 0,C 180,E1 -16651.393,E2 -16651.393} C_VEL
LIN {X 0,Y 289.429,Z 399.713,A -85,B 0,C 180,E1 -16652.785,E2 -16652.785} C_VEL
LIN {X 0,Y 289.434,Z 398.632,A -85,B 0,C 180,E1 -16655.402,E2 -16655.402} C_VEL
LIN {X 0,Y 289.641,Z 397.284,A -85,B 0,C 180,E1 -16656.97,E2 -16656.97} C_VEL
LIN {X 0,Y 290.131,Z 394.631,A -85,B 0,C 180,E1 -16659.06,E2 -16659.06} C_VEL
LIN {X 0,Y 290.873,Z 390.96,A -85,B 0,C 180,E1 -16661.146,E2 -16661.146} C_VEL
LIN {X 0,Y 291.924,Z 386.193,A -85,B 0,C 180,E1 -16663.222,E2 -16663.222} C_VEL
LIN {X 0,Y 293.546,Z 380.166,A -85,B 0,C 180,E1 -16665.271,E2 -16665.271} C_VEL
LIN {X 0,Y 295.314,Z 372.705,A -85,B 0,C 180,E1 -16667.307,E2 -16667.307} C_VEL
LIN {X 0,Y 297.005,Z 365.156,A -85,B 0,C 180,E1 -16668.991,E2 -16668.991} C_VEL
LIN {X 0,Y 299.278,Z 355.141,A -85,B 0,C 180,E1 -16670.806,E2 -16670.806} C_VEL
LIN {X 0,Y 301.785,Z 343.769,A -85,B 0,C 180,E1 -16672.418,E2 -16672.418} C_VEL
LIN {X 0,Y 303.901,Z 332.501,A -85,B 0,C 180,E1 -16673.693,E2 -16673.693} C_VEL
LIN {X 0,Y 305.833,Z 319.931,A -85,B 0,C 180,E1 -16674.797,E2 -16674.797} C_VEL
LIN {X 0,Y 307.73,Z 306.638,A -85,B 0,C 180,E1 -16675.627,E2 -16675.627} C_VEL
LIN {X 0,Y 308.893,Z 293.706,A -85,B 0,C 180,E1 -16676.203,E2 -16676.203} C_VEL
LIN {X 0,Y 312.305,Z 232.787,A -85,B 0,C 180,E1 -16678.082,E2 -16678.082} C_VEL
LIN {X 0,Y 310.301,Z 218.533,A -85,B 0,C 180,E1 -16678.958,E2 -16678.958} C_VEL
LIN {X 0,Y 308.433,Z 209.148,A -85,B 0,C 180,E1 -16679.634,E2 -16679.634} C_VEL
LIN {X 0,Y 303.332,Z 197.922,A -85,B 0,C 180,E1 -16680.989,E2 -16680.989} C_VEL
LIN {X 0,Y 299.08,Z 189.815,A -85,B 0,C 180,E1 -16682.147,E2 -16682.147} C_VEL
LIN {X 0,Y 296.607,Z 185.214,A -85,B 0,C 180,E1 -16682.879,E2 -16682.879} C_VEL
LIN {X 0,Y 294.828,Z 178.372,A -85,B 0,C 180,E1 -16685.857,E2 -16685.857} C_VEL
LIN {X 0,Y 292.84,Z 171.96,A -85,B 0,C 180,E1 -16689.037,E2 -16689.037} C_VEL
LIN {X 0,Y 291.283,Z 167.201,A -85,B 0,C 180,E1 -16691.731,E2 -16691.731} C_VEL
LIN {X 0,Y 291.285,Z 167.194,A -85,B 0,C 180,E1 -16695.597,E2 -16695.597} C_VEL
LIN {X 0,Y 291.303,Z 167.19,A -85,B 0,C 180,E1 -16699.353,E2 -16699.353} C_VEL
LIN {X 0,Y 291.389,Z 167.186,A -85,B 0,C 180,E1 -16702.917,E2 -16702.917} C_VEL
LIN {X 0,Y 291.347,Z 167.189,A -85,B 0,C 180,E1 -16706.302,E2 -16706.302} C_VEL
LIN {X 0,Y 291.368,Z 167.19,A -85,B 0,C 180,E1 -16710.269,E2 -16710.269} C_VEL
LIN {X 0,Y 291.35,Z 167.186,A -85,B 0,C 180,E1 -16714.266,E2 -16714.266} C_VEL
LIN {X 0,Y 291.354,Z 167.187,A -85,B 0,C 180,E1 -16717.297,E2 -16717.297} C_VEL
LIN {X 0,Y 291.389,Z 167.187,A -85,B 0,C 180,E1 -16720.266,E2 -16720.266} C_VEL
LIN {X 0,Y 291.478,Z 167.177,A -85,B 0,C 180,E1 -16724.683,E2 -16724.683} C_VEL
LIN {X 0,Y 291.532,Z 167.173,A -85,B 0,C 180,E1 -16728.881,E2 -16728.881} C_VEL
LIN {X 0,Y 291.602,Z 167.294,A -85,B 0,C 180,E1 -16730.287,E2 -16730.287} C_VEL
LIN {X 0,Y 293.345,Z 172.295,A -85,B 0,C 180,E1 -16733.12,E2 -16733.12} C_VEL
LIN {X 0,Y 294.201,Z 175.572,A -85,B 0,C 180,E1 -16734.689,E2 -16734.689} C_VEL
LIN {X 0,Y 297.224,Z 180.242,A -85,B 0,C 180,E1 -16735.559,E2 -16735.559} C_VEL
LIN {X 0,Y 301.072,Z 186.284,A -85,B 0,C 180,E1 -16736.605,E2 -16736.605} C_VEL
LIN {X 0,Y 307.006,Z 197.068,A -85,B 0,C 180,E1 -16738.144,E2 -16738.144} C_VEL
LIN {X 0,Y 310.981,Z 205.82,A -85,B 0,C 180,E1 -16739.156,E2 -16739.156} C_VEL
LIN {X 0,Y 313.417,Z 211.447,A -85,B 0,C 180,E1 -16739.758,E2 -16739.758} C_VEL
LIN {X 0,Y 309.077,Z 284.079,A -85,B 0,C 180,E1 -16742.022,E2 -16742.022} C_VEL
LIN {X 0,Y 307.808,Z 297.527,A -85,B 0,C 180,E1 -16742.699,E2 -16742.699} C_VEL
LIN {X 0,Y 306.172,Z 310.259,A -85,B 0,C 180,E1 -16743.62,E2 -16743.62} C_VEL
LIN {X 0,Y 304.373,Z 321.993,A -85,B 0,C 180,E1 -16744.747,E2 -16744.747} C_VEL
LIN {X 0,Y 302.192,Z 333.638,A -85,B 0,C 180,E1 -16746.175,E2 -16746.175} C_VEL
LIN {X 0,Y 299.787,Z 344.767,A -85,B 0,C 180,E1 -16747.917,E2 -16747.917} C_VEL
LIN {X 0,Y 297.834,Z 352.96,A -85,B 0,C 180,E1 -16749.508,E2 -16749.508} C_VEL
LIN {X 0,Y 296.011,Z 360.497,A -85,B 0,C 180,E1 -16751.296,E2 -16751.296} C_VEL
LIN {X 0,Y 294.097,Z 367.806,A -85,B 0,C 180,E1 -16753.474,E2 -16753.474} C_VEL
LIN {X 0,Y 292.373,Z 374.202,A -85,B 0,C 180,E1 -16755.944,E2 -16755.944} C_VEL
LIN {X 0,Y 291.159,Z 378.639,A -85,B 0,C 180,E1 -16758.289,E2 -16758.289} C_VEL
LIN {X 0,Y 290.603,Z 380.758,A -85,B 0,C 180,E1 -16759.791,E2 -16759.791} C_VEL
LIN {X 0,Y 290.096,Z 382.423,A -85,B 0,C 180,E1 -16761.309,E2 -16761.309} C_VEL
LIN {X 0,Y 289.736,Z 383.529,A -85,B 0,C 180,E1 -16762.837,E2 -16762.837} C_VEL
LIN {X 0,Y 289.434,Z 384.173,A -85,B 0,C 180,E1 -16764.381,E2 -16764.381} C_VEL
LIN {X 0,Y 289.258,Z 384.284,A -85,B 0,C 180,E1 -16765.974,E2 -16765.974} C_VEL
LIN {X 0,Y 289.134,Z 383.874,A -85,B 0,C 180,E1 -16767.506,E2 -16767.506} C_VEL
LIN {X 0,Y 289.143,Z 382.944,A -85,B 0,C 180,E1 -16769.087,E2 -16769.087} C_VEL
LIN {X 0,Y 289.321,Z 380.053,A -85,B 0,C 180,E1 -16771.765,E2 -16771.765} C_VEL
LIN {X 0,Y 289.667,Z 376.517,A -85,B 0,C 180,E1 -16773.921,E2 -16773.921} C_VEL
LIN {X 0,Y 290.046,Z 371.321,A -85,B 0,C 180,E1 -16776.264,E2 -16776.264} C_VEL
LIN {X 0,Y 290.706,Z 364.789,A -85,B 0,C 180,E1 -16778.501,E2 -16778.501} C_VEL
LIN {X 0,Y 291.547,Z 357.033,A -85,B 0,C 180,E1 -16780.607,E2 -16780.607} C_VEL
LIN {X 0,Y 292.525,Z 348.334,A -85,B 0,C 180,E1 -16782.51,E2 -16782.51} C_VEL
LIN {X 0,Y 293.472,Z 338.895,A -85,B 0,C 180,E1 -16784.18,E2 -16784.18} C_VEL
LIN {X 0,Y 294.736,Z 327.098,A -85,B 0,C 180,E1 -16785.856,E2 -16785.856} C_VEL
LIN {X 0,Y 295.822,Z 316.399,A -85,B 0,C 180,E1 -16787.057,E2 -16787.057} C_VEL
LIN {X 0,Y 296.872,Z 303.217,A -85,B 0,C 180,E1 -16788.205,E2 -16788.205} C_VEL
LIN {X 0,Y 297.654,Z 289.951,A -85,B 0,C 180,E1 -16789.049,E2 -16789.049} C_VEL
LIN {X 0,Y 298.341,Z 275.699,A -85,B 0,C 180,E1 -16789.635,E2 -16789.635} C_VEL
LIN {X 0,Y 300.57,Z 204.512,A -85,B 0,C 180,E1 -16791.71,E2 -16791.71} C_VEL
LIN {X 0,Y 298.116,Z 190.555,A -85,B 0,C 180,E1 -16792.295,E2 -16792.295} C_VEL
LIN {X 0,Y 292.544,Z 172.819,A -85,B 0,C 180,E1 -16793.247,E2 -16793.247} C_VEL
LIN {X 0,Y 291.432,Z 167.181,A -85,B 0,C 180,E1 -16795.195,E2 -16795.195} C_VEL
LIN {X 0,Y 291.371,Z 167.189,A -85,B 0,C 180,E1 -16797.949,E2 -16797.949} C_VEL
LIN {X 0,Y 291.32,Z 167.195,A -85,B 0,C 180,E1 -16801.15,E2 -16801.15} C_VEL
LIN {X 0,Y 291.347,Z 167.196,A -85,B 0,C 180,E1 -16804.264,E2 -16804.264} C_VEL
LIN {X 0,Y 291.354,Z 167.19,A -85,B 0,C 180,E1 -16807.296,E2 -16807.296} C_VEL
LIN {X 0,Y 291.389,Z 167.191,A -85,B 0,C 180,E1 -16810.264,E2 -16810.264} C_VEL
LIN {X 0,Y 291.479,Z 167.176,A -85,B 0,C 180,E1 -16814.682,E2 -16814.682} C_VEL
LIN {X 0,Y 291.531,Z 167.168,A -85,B 0,C 180,E1 -16818.879,E2 -16818.879} C_VEL
LIN {X 0,Y 291.656,Z 167.155,A -85,B 0,C 180,E1 -16821.686,E2 -16821.686} C_VEL
LIN {X 0,Y 291.6,Z 167.16,A -85,B 0,C 180,E1 -16824.467,E2 -16824.467} C_VEL
LIN {X 0,Y 291.874,Z 167.125,A -85,B 0,C 180,E1 -16828.619,E2 -16828.619} C_VEL
LIN {X 0,Y 291.874,Z 167.126,A -85,B 0,C 180,E1 -16831.379,E2 -16831.379} C_VEL
LIN {X 0,Y 291.688,Z 167.148,A -85,B 0,C 180,E1 -16836.918,E2 -16836.918} C_VEL
LIN {X 0,Y 291.57,Z 167.167,A -85,B 0,C 180,E1 -16839.713,E2 -16839.713} C_VEL
LIN {X 0,Y 291.483,Z 167.175,A -85,B 0,C 180,E1 -16843.951,E2 -16843.951} C_VEL
LIN {X 0,Y 291.403,Z 167.184,A -85,B 0,C 180,E1 -16846.822,E2 -16846.822} C_VEL
LIN {X 0,Y 291.392,Z 167.187,A -85,B 0,C 180,E1 -16849.841,E2 -16849.841} C_VEL
LIN {X 0,Y 291.326,Z 167.193,A -85,B 0,C 180,E1 -16854.21,E2 -16854.21} C_VEL
LIN {X 0,Y 291.349,Z 167.195,A -85,B 0,C 180,E1 -16857.277,E2 -16857.277} C_VEL
LIN {X 0,Y 291.317,Z 167.195,A -85,B 0,C 180,E1 -16860.438,E2 -16860.438} C_VEL
LIN {X 0,Y 291.342,Z 167.191,A -85,B 0,C 180,E1 -16863.697,E2 -16863.697} C_VEL
LIN {X 0,Y 291.357,Z 167.193,A -85,B 0,C 180,E1 -16867.248,E2 -16867.248} C_VEL
LIN {X 0,Y 291.298,Z 167.199,A -85,B 0,C 180,E1 -16870.647,E2 -16870.647} C_VEL
LIN {X 0,Y 291.278,Z 167.2,A -85,B 0,C 180,E1 -16874.402,E2 -16874.402} C_VEL
LIN {X 0,Y 291.291,Z 167.2,A -85,B 0,C 180,E1 -16878.41,E2 -16878.41} C_VEL
LIN {X 0,Y 291.33,Z 167.194,A -85,B 0,C 180,E1 -16881.154,E2 -16881.154} C_VEL
LIN {X 0,Y 291.351,Z 167.195,A -85,B 0,C 180,E1 -16884.624,E2 -16884.624} C_VEL
LIN {X 0,Y 291.361,Z 167.189,A -85,B 0,C 180,E1 -16887.949,E2 -16887.949} C_VEL
LIN {X 0,Y 291.336,Z 167.193,A -85,B 0,C 180,E1 -16891.153,E2 -16891.153} C_VEL
LIN {X 0,Y 291.336,Z 167.195,A -85,B 0,C 180,E1 -16894.264,E2 -16894.264} C_VEL
LIN {X 0,Y 291.339,Z 167.195,A -85,B 0,C 180,E1 -16896.296,E2 -16896.296} C_VEL
LIN {X 0,Y 290.716,Z 167.277,A -85,B 0,C 180,E1 -16897.45,E2 -16897.45} C_VEL
LIN {X 0,Y 287.843,Z 167.631,A -85,B 0,C 180,E1 -16899.329,E2 -16899.329} C_VEL
LIN {X 0,Y 285.399,Z 167.933,A -85,B 0,C 180,E1 -16900.855,E2 -16900.855} C_VEL
LIN {X 0,Y 284.385,Z 168.061,A -85,B 0,C 180,E1 -16902.038,E2 -16902.038} C_VEL
LIN {X 0,Y 284.323,Z 168.065,A -85,B 0,C 180,E1 -16902.439,E2 -16902.439} C_VEL
LIN {X 0,Y 284.411,Z 168.055,A -85,B 0,C 180,E1 -16905.693,E2 -16905.693} C_VEL
LIN {X 0,Y 284.507,Z 168.047,A -85,B 0,C 180,E1 -16910.042,E2 -16910.042} C_VEL
LIN {X 0,Y 284.635,Z 168.026,A -85,B 0,C 180,E1 -16912.908,E2 -16912.908} C_VEL
LIN {X 0,Y 284.83,Z 168.003,A -85,B 0,C 180,E1 -16918.586,E2 -16918.586} C_VEL
LIN {X 0,Y 284.83,Z 168.003,A -85,B 0,C 180,E1 -16921.414,E2 -16921.414} C_VEL
LIN {X 0,Y 284.634,Z 168.027,A -85,B 0,C 180,E1 -16927.091,E2 -16927.091} C_VEL
LIN {X 0,Y 284.506,Z 168.045,A -85,B 0,C 180,E1 -16929.957,E2 -16929.957} C_VEL
LIN {X 0,Y 284.41,Z 168.056,A -85,B 0,C 180,E1 -16934.306,E2 -16934.306} C_VEL
LIN {X 0,Y 284.308,Z 168.067,A -85,B 0,C 180,E1 -16938.745,E2 -16938.745} C_VEL
LIN {X 0,Y 284.288,Z 168.073,A -85,B 0,C 180,E1 -16941.766,E2 -16941.766} C_VEL
LIN {X 0,Y 284.276,Z 168.073,A -85,B 0,C 180,E1 -16944.852,E2 -16944.852} C_VEL
LIN {X 0,Y 284.273,Z 168.072,A -85,B 0,C 180,E1 -16948.017,E2 -16948.017} C_VEL
LIN {X 0,Y 284.278,Z 168.076,A -85,B 0,C 180,E1 -16951.276,E2 -16951.276} C_VEL
LIN {X 0,Y 284.33,Z 168.067,A -85,B 0,C 180,E1 -16955.347,E2 -16955.347} C_VEL
LIN {X 0,Y 284.291,Z 168.069,A -85,B 0,C 180,E1 -16958.172,E2 -16958.172} C_VEL
LIN {X 0,Y 284.231,Z 168.077,A -85,B 0,C 180,E1 -16962.118,E2 -16962.118} C_VEL
LIN {X 0,Y 284.232,Z 168.078,A -85,B 0,C 180,E1 -16966.187,E2 -16966.187} C_VEL
LIN {X 0,Y 284.278,Z 168.072,A -85,B 0,C 180,E1 -16970.031,E2 -16970.031} C_VEL
LIN {X 0,Y 284.316,Z 168.067,A -85,B 0,C 180,E1 -16973.613,E2 -16973.613} C_VEL
LIN {X 0,Y 284.339,Z 168.158,A -85,B 0,C 180,E1 -16978.005,E2 -16978.005} C_VEL
LIN {X 0,Y 286.934,Z 181.235,A -85,B 0,C 180,E1 -16982.267,E2 -16982.267} C_VEL
LIN {X 0,Y 288.085,Z 188.408,A -85,B 0,C 180,E1 -16984.507,E2 -16984.507} C_VEL
LIN {X 0,Y 293.294,Z 230.983,A -85,B 0,C 180,E1 -16986.213,E2 -16986.213} C_VEL
LIN {X 0,Y 291.096,Z 297.766,A -85,B 0,C 180,E1 -16988.258,E2 -16988.258} C_VEL
LIN {X 0,Y 290.257,Z 311.834,A -85,B 0,C 180,E1 -16988.984,E2 -16988.984} C_VEL
LIN {X 0,Y 289.172,Z 324.428,A -85,B 0,C 180,E1 -16989.924,E2 -16989.924} C_VEL
LIN {X 0,Y 288.021,Z 336.65,A -85,B 0,C 180,E1 -16991.138,E2 -16991.138} C_VEL
LIN {X 0,Y 286.776,Z 347.683,A -85,B 0,C 180,E1 -16992.531,E2 -16992.531} C_VEL
LIN {X 0,Y 285.635,Z 358.718,A -85,B 0,C 180,E1 -16994.298,E2 -16994.298} C_VEL
LIN {X 0,Y 284.584,Z 367.679,A -85,B 0,C 180,E1 -16996.069,E2 -16996.069} C_VEL
LIN {X 0,Y 283.571,Z 376.355,A -85,B 0,C 180,E1 -16998.203,E2 -16998.203} C_VEL
LIN {X 0,Y 282.961,Z 383.309,A -85,B 0,C 180,E1 -17000.35,E2 -17000.35} C_VEL
LIN {X 0,Y 282.573,Z 389.638,A -85,B 0,C 180,E1 -17002.858,E2 -17002.858} C_VEL
LIN {X 0,Y 282.427,Z 392.801,A -85,B 0,C 180,E1 -17004.487,E2 -17004.487} C_VEL
LIN {X 0,Y 282.368,Z 394.781,A -85,B 0,C 180,E1 -17005.719,E2 -17005.719} C_VEL
LIN {X 0,Y 282.401,Z 396.632,A -85,B 0,C 180,E1 -17007.148,E2 -17007.148} C_VEL
LIN {X 0,Y 282.346,Z 397.992,A -85,B 0,C 180,E1 -17008.575,E2 -17008.575} C_VEL
LIN {X 0,Y 282.358,Z 398.936,A -85,B 0,C 180,E1 -17010.001,E2 -17010.001} C_VEL
LIN {X 0,Y 282.33,Z 399.463,A -85,B 0,C 180,E1 -17011.428,E2 -17011.428} C_VEL
LIN {X 0,Y 282.335,Z 399.532,A -85,B 0,C 180,E1 -17012.855,E2 -17012.855} C_VEL
LIN {X 0,Y 282.355,Z 398.649,A -85,B 0,C 180,E1 -17015.361,E2 -17015.361} C_VEL
LIN {X 0,Y 282.582,Z 397.279,A -85,B 0,C 180,E1 -17017.145,E2 -17017.145} C_VEL
LIN {X 0,Y 283.103,Z 394.72,A -85,B 0,C 180,E1 -17019.287,E2 -17019.287} C_VEL
LIN {X 0,Y 283.897,Z 391.153,A -85,B 0,C 180,E1 -17021.424,E2 -17021.424} C_VEL
LIN {X 0,Y 285.013,Z 386.498,A -85,B 0,C 180,E1 -17023.549,E2 -17023.549} C_VEL
LIN {X 0,Y 287.024,Z 379.475,A -85,B 0,C 180,E1 -17025.991,E2 -17025.991} C_VEL
LIN {X 0,Y 288.901,Z 371.949,A -85,B 0,C 180,E1 -17028.07,E2 -17028.07} C_VEL
LIN {X 0,Y 290.723,Z 364.363,A -85,B 0,C 180,E1 -17029.783,E2 -17029.783} C_VEL
LIN {X 0,Y 293.249,Z 354.201,A -85,B 0,C 180,E1 -17031.623,E2 -17031.623} C_VEL
LIN {X 0,Y 295.856,Z 342.665,A -85,B 0,C 180,E1 -17033.262,E2 -17033.262} C_VEL
LIN {X 0,Y 298.117,Z 331.171,A -85,B 0,C 180,E1 -17034.552,E2 -17034.552} C_VEL
LIN {X 0,Y 300.203,Z 318.248,A -85,B 0,C 180,E1 -17035.666,E2 -17035.666} C_VEL
LIN {X 0,Y 301.991,Z 306.045,A -85,B 0,C 180,E1 -17036.43,E2 -17036.43} C_VEL
LIN {X 0,Y 303.211,Z 293.103,A -85,B 0,C 180,E1 -17037.012,E2 -17037.012} C_VEL
LIN {X 0,Y 306.736,Z 234.208,A -85,B 0,C 180,E1 -17038.867,E2 -17038.867} C_VEL
LIN {X 0,Y 304.946,Z 220.828,A -85,B 0,C 180,E1 -17039.71,E2 -17039.71} C_VEL
LIN {X 0,Y 303.313,Z 212.29,A -85,B 0,C 180,E1 -17040.363,E2 -17040.363} C_VEL
LIN {X 0,Y 297.521,Z 199.557,A -85,B 0,C 180,E1 -17041.989,E2 -17041.989} C_VEL
LIN {X 0,Y 293.92,Z 193.037,A -85,B 0,C 180,E1 -17043.03,E2 -17043.03} C_VEL
LIN {X 0,Y 292.049,Z 189.702,A -85,B 0,C 180,E1 -17043.594,E2 -17043.594} C_VEL
LIN {X 0,Y 289.532,Z 185.228,A -85,B 0,C 180,E1 -17044.381,E2 -17044.381} C_VEL
LIN {X 0,Y 289.175,Z 184,A -85,B 0,C 180,E1 -17044.836,E2 -17044.836} C_VEL
LIN {X 0,Y 287.066,Z 176.709,A -85,B 0,C 180,E1 -17048.424,E2 -17048.424} C_VEL
LIN {X 0,Y 285.221,Z 170.971,A -85,B 0,C 180,E1 -17051.706,E2 -17051.706} C_VEL
LIN {X 0,Y 284.246,Z 168.073,A -85,B 0,C 180,E1 -17053.59,E2 -17053.59} C_VEL
LIN {X 0,Y 284.24,Z 168.073,A -85,B 0,C 180,E1 -17057.884,E2 -17057.884} C_VEL
LIN {X 0,Y 284.298,Z 168.063,A -85,B 0,C 180,E1 -17061.829,E2 -17061.829} C_VEL
LIN {X 0,Y 284.311,Z 168.071,A -85,B 0,C 180,E1 -17065.351,E2 -17065.351} C_VEL
LIN {X 0,Y 284.288,Z 168.068,A -85,B 0,C 180,E1 -17068.725,E2 -17068.725} C_VEL
LIN {X 0,Y 284.284,Z 168.066,A -85,B 0,C 180,E1 -17071.985,E2 -17071.985} C_VEL
LIN {X 0,Y 284.302,Z 168.066,A -85,B 0,C 180,E1 -17076.158,E2 -17076.158} C_VEL
LIN {X 0,Y 284.338,Z 168.063,A -85,B 0,C 180,E1 -17079.929,E2 -17079.929} C_VEL
LIN {X 0,Y 284.419,Z 168.055,A -85,B 0,C 180,E1 -17084.517,E2 -17084.517} C_VEL
LIN {X 0,Y 284.494,Z 168.199,A -85,B 0,C 180,E1 -17088.421,E2 -17088.421} C_VEL
LIN {X 0,Y 286.294,Z 173.05,A -85,B 0,C 180,E1 -17091.53,E2 -17091.53} C_VEL
LIN {X 0,Y 287.212,Z 175.907,A -85,B 0,C 180,E1 -17093.092,E2 -17093.092} C_VEL
LIN {X 0,Y 290.173,Z 180.589,A -85,B 0,C 180,E1 -17094.057,E2 -17094.057} C_VEL
LIN {X 0,Y 297.194,Z 191.669,A -85,B 0,C 180,E1 -17096.104,E2 -17096.104} C_VEL
LIN {X 0,Y 302.567,Z 201.719,A -85,B 0,C 180,E1 -17097.568,E2 -17097.568} C_VEL
LIN {X 0,Y 306.494,Z 210.697,A -85,B 0,C 180,E1 -17098.645,E2 -17098.645} C_VEL
LIN {X 0,Y 307.864,Z 213.871,A -85,B 0,C 180,E1 -17098.996,E2 -17098.996} C_VEL
LIN {X 0,Y 303.429,Z 283.788,A -85,B 0,C 180,E1 -17101.208,E2 -17101.208} C_VEL
LIN {X 0,Y 302.042,Z 297.417,A -85,B 0,C 180,E1 -17101.9,E2 -17101.9} C_VEL
LIN {X 0,Y 300.318,Z 310.323,A -85,B 0,C 180,E1 -17102.851,E2 -17102.851} C_VEL
LIN {X 0,Y 298.314,Z 322.584,A -85,B 0,C 180,E1 -17104.053,E2 -17104.053} C_VEL
LIN {X 0,Y 296.138,Z 333.739,A -85,B 0,C 180,E1 -17105.448,E2 -17105.448} C_VEL
LIN {X 0,Y 293.833,Z 343.894,A -85,B 0,C 180,E1 -17107.041,E2 -17107.041} C_VEL
LIN {X 0,Y 291.55,Z 352.757,A -85,B 0,C 180,E1 -17108.756,E2 -17108.756} C_VEL
LIN {X 0,Y 289.36,Z 361.312,A -85,B 0,C 180,E1 -17110.85,E2 -17110.85} C_VEL
LIN {X 0,Y 287.311,Z 368.498,A -85,B 0,C 180,E1 -17113.078,E2 -17113.078} C_VEL
LIN {X 0,Y 285.917,Z 373.327,A -85,B 0,C 180,E1 -17114.958,E2 -17114.958} C_VEL
LIN {X 0,Y 284.563,Z 377.884,A -85,B 0,C 180,E1 -17117.24,E2 -17117.24} C_VEL
LIN {X 0,Y 283.58,Z 381.324,A -85,B 0,C 180,E1 -17119.648,E2 -17119.648} C_VEL
LIN {X 0,Y 282.854,Z 383.377,A -85,B 0,C 180,E1 -17121.883,E2 -17121.883} C_VEL
LIN {X 0,Y 282.518,Z 384.19,A -85,B 0,C 180,E1 -17123.455,E2 -17123.455} C_VEL
LIN {X 0,Y 282.145,Z 384.41,A -85,B 0,C 180,E1 -17126.266,E2 -17126.266} C_VEL
LIN {X 0,Y 282.032,Z 383.579,A -85,B 0,C 180,E1 -17128.26,E2 -17128.26} C_VEL
LIN {X 0,Y 282.045,Z 382.315,A -85,B 0,C 180,E1 -17129.892,E2 -17129.892} C_VEL
LIN {X 0,Y 282.311,Z 379.552,A -85,B 0,C 180,E1 -17132.174,E2 -17132.174} C_VEL
LIN {X 0,Y 282.583,Z 376.418,A -85,B 0,C 180,E1 -17134.028,E2 -17134.028} C_VEL
LIN {X 0,Y 283.016,Z 370.687,A -85,B 0,C 180,E1 -17136.583,E2 -17136.583} C_VEL
LIN {X 0,Y 283.676,Z 364.503,A -85,B 0,C 180,E1 -17138.703,E2 -17138.703} C_VEL
LIN {X 0,Y 284.534,Z 356.534,A -85,B 0,C 180,E1 -17140.886,E2 -17140.886} C_VEL
LIN {X 0,Y 285.535,Z 347.751,A -85,B 0,C 180,E1 -17142.811,E2 -17142.811} C_VEL
LIN {X 0,Y 286.663,Z 337.148,A -85,B 0,C 180,E1 -17144.684,E2 -17144.684} C_VEL
LIN {X 0,Y 287.749,Z 327.227,A -85,B 0,C 180,E1 -17146.098,E2 -17146.098} C_VEL
LIN {X 0,Y 288.906,Z 315.983,A -85,B 0,C 180,E1 -17147.381,E2 -17147.381} C_VEL
LIN {X 0,Y 290.024,Z 302.538,A -85,B 0,C 180,E1 -17148.565,E2 -17148.565} C_VEL
LIN {X 0,Y 290.788,Z 289.32,A -85,B 0,C 180,E1 -17149.406,E2 -17149.406} C_VEL
LIN {X 0,Y 291.508,Z 275.085,A -85,B 0,C 180,E1 -17149.992,E2 -17149.992} C_VEL
LIN {X 0,Y 293.801,Z 205.645,A -85,B 0,C 180,E1 -17152.077,E2 -17152.077} C_VEL
LIN {X 0,Y 291.628,Z 192.924,A -85,B 0,C 180,E1 -17152.618,E2 -17152.618} C_VEL
LIN {X 0,Y 285.357,Z 173.005,A -85,B 0,C 180,E1 -17153.71,E2 -17153.71} C_VEL
LIN {X 0,Y 284.383,Z 168.059,A -85,B 0,C 180,E1 -17155.467,E2 -17155.467} C_VEL
LIN {X 0,Y 284.314,Z 168.072,A -85,B 0,C 180,E1 -17160.37,E2 -17160.37} C_VEL
LIN {X 0,Y 284.3,Z 168.069,A -85,B 0,C 180,E1 -17163.578,E2 -17163.578} C_VEL
LIN {X 0,Y 284.312,Z 168.069,A -85,B 0,C 180,E1 -17166.701,E2 -17166.701} C_VEL
LIN {X 0,Y 284.339,Z 168.066,A -85,B 0,C 180,E1 -17169.927,E2 -17169.927} C_VEL
LIN {X 0,Y 284.419,Z 168.056,A -85,B 0,C 180,E1 -17174.515,E2 -17174.515} C_VEL
LIN {X 0,Y 284.463,Z 168.05,A -85,B 0,C 180,E1 -17178.599,E2 -17178.599} C_VEL
LIN {X 0,Y 284.613,Z 168.031,A -85,B 0,C 180,E1 -17181.479,E2 -17181.479} C_VEL
LIN {X 0,Y 284.57,Z 168.037,A -85,B 0,C 180,E1 -17184.329,E2 -17184.329} C_VEL
LIN {X 0,Y 284.841,Z 168.001,A -85,B 0,C 180,E1 -17188.585,E2 -17188.585} C_VEL
LIN {X 0,Y 284.841,Z 168.002,A -85,B 0,C 180,E1 -17191.413,E2 -17191.413} C_VEL
LIN {X 0,Y 284.644,Z 168.026,A -85,B 0,C 180,E1 -17197.09,E2 -17197.09} C_VEL
LIN {X 0,Y 284.516,Z 168.044,A -85,B 0,C 180,E1 -17199.956,E2 -17199.956} C_VEL
LIN {X 0,Y 284.42,Z 168.054,A -85,B 0,C 180,E1 -17204.305,E2 -17204.305} C_VEL
LIN {X 0,Y 284.317,Z 168.067,A -85,B 0,C 180,E1 -17208.743,E2 -17208.743} C_VEL
LIN {X 0,Y 284.296,Z 168.071,A -85,B 0,C 180,E1 -17211.764,E2 -17211.764} C_VEL
LIN {X 0,Y 284.283,Z 168.072,A -85,B 0,C 180,E1 -17214.85,E2 -17214.85} C_VEL
LIN {X 0,Y 284.28,Z 168.071,A -85,B 0,C 180,E1 -17218.015,E2 -17218.015} C_VEL
LIN {X 0,Y 284.284,Z 168.074,A -85,B 0,C 180,E1 -17221.274,E2 -17221.274} C_VEL
LIN {X 0,Y 284.335,Z 168.067,A -85,B 0,C 180,E1 -17225.345,E2 -17225.345} C_VEL
LIN {X 0,Y 284.295,Z 168.069,A -85,B 0,C 180,E1 -17228.17,E2 -17228.17} C_VEL
LIN {X 0,Y 284.234,Z 168.076,A -85,B 0,C 180,E1 -17232.116,E2 -17232.116} C_VEL
LIN {X 0,Y 284.234,Z 168.078,A -85,B 0,C 180,E1 -17236.184,E2 -17236.184} C_VEL
LIN {X 0,Y 284.279,Z 168.071,A -85,B 0,C 180,E1 -17240.028,E2 -17240.028} C_VEL
LIN {X 0,Y 284.317,Z 168.067,A -85,B 0,C 180,E1 -17243.611,E2 -17243.611} C_VEL
LIN {X 0,Y 284.301,Z 168.069,A -85,B 0,C 180,E1 -17247.189,E2 -17247.189} C_VEL
LIN {X 0,Y 284.331,Z 168.067,A -85,B 0,C 180,E1 -17250.372,E2 -17250.372} C_VEL
LIN {X 0,Y 284.291,Z 168.07,A -85,B 0,C 180,E1 -17253.577,E2 -17253.577} C_VEL
LIN {X 0,Y 284.301,Z 168.07,A -85,B 0,C 180,E1 -17256.701,E2 -17256.701} C_VEL
LIN {X 0,Y 284.328,Z 168.067,A -85,B 0,C 180,E1 -17259.927,E2 -17259.927} C_VEL
LIN {X 0,Y 284.323,Z 168.065,A -85,B 0,C 180,E1 -17262.439,E2 -17262.439} C_VEL
LIN {X 0,Y 283.716,Z 168.146,A -85,B 0,C 180,E1 -17263.621,E2 -17263.621} C_VEL
LIN {X 0,Y 280.911,Z 168.5,A -85,B 0,C 180,E1 -17265.548,E2 -17265.548} C_VEL
LIN {X 0,Y 278.503,Z 168.798,A -85,B 0,C 180,E1 -17267.114,E2 -17267.114} C_VEL
LIN {X 0,Y 277.474,Z 168.923,A -85,B 0,C 180,E1 -17268.326,E2 -17268.326} C_VEL
LIN {X 0,Y 277.394,Z 168.93,A -85,B 0,C 180,E1 -17268.737,E2 -17268.737} C_VEL
LIN {X 0,Y 277.563,Z 168.908,A -85,B 0,C 180,E1 -17271.261,E2 -17271.261} C_VEL
LIN {X 0,Y 277.531,Z 168.915,A -85,B 0,C 180,E1 -17274.186,E2 -17274.186} C_VEL
LIN {X 0,Y 277.797,Z 168.88,A -85,B 0,C 180,E1 -17278.55,E2 -17278.55} C_VEL
LIN {X 0,Y 277.797,Z 168.88,A -85,B 0,C 180,E1 -17281.449,E2 -17281.449} C_VEL
LIN {X 0,Y 277.593,Z 168.905,A -85,B 0,C 180,E1 -17287.272,E2 -17287.272} C_VEL
LIN {X 0,Y 277.446,Z 168.922,A -85,B 0,C 180,E1 -17290.213,E2 -17290.213} C_VEL
LIN {X 0,Y 277.363,Z 168.933,A -85,B 0,C 180,E1 -17294.678,E2 -17294.678} C_VEL
LIN {X 0,Y 277.268,Z 168.946,A -85,B 0,C 180,E1 -17299.239,E2 -17299.239} C_VEL
LIN {X 0,Y 277.248,Z 168.948,A -85,B 0,C 180,E1 -17303.928,E2 -17303.928} C_VEL
LIN {X 0,Y 277.259,Z 168.949,A -85,B 0,C 180,E1 -17307.482,E2 -17307.482} C_VEL
LIN {X 0,Y 277.241,Z 168.948,A -85,B 0,C 180,E1 -17310.473,E2 -17310.473} C_VEL
LIN {X 0,Y 277.239,Z 168.948,A -85,B 0,C 180,E1 -17313.897,E2 -17313.897} C_VEL
LIN {X 0,Y 277.248,Z 168.949,A -85,B 0,C 180,E1 -17317.472,E2 -17317.472} C_VEL
LIN {X 0,Y 277.178,Z 168.959,A -85,B 0,C 180,E1 -17321.242,E2 -17321.242} C_VEL
LIN {X 0,Y 277.168,Z 168.961,A -85,B 0,C 180,E1 -17325.233,E2 -17325.233} C_VEL
LIN {X 0,Y 277.179,Z 168.96,A -85,B 0,C 180,E1 -17328.76,E2 -17328.76} C_VEL
LIN {X 0,Y 277.25,Z 168.95,A -85,B 0,C 180,E1 -17332.53,E2 -17332.53} C_VEL
LIN {X 0,Y 277.242,Z 168.949,A -85,B 0,C 180,E1 -17336.105,E2 -17336.105} C_VEL
LIN {X 0,Y 277.291,Z 169.056,A -85,B 0,C 180,E1 -17337.709,E2 -17337.709} C_VEL
LIN {X 0,Y 279.742,Z 181.31,A -85,B 0,C 180,E1 -17341.81,E2 -17341.81} C_VEL
LIN {X 0,Y 280.989,Z 188.192,A -85,B 0,C 180,E1 -17344.03,E2 -17344.03} C_VEL
LIN {X 0,Y 282.153,Z 196.021,A -85,B 0,C 180,E1 -17344.391,E2 -17344.391} C_VEL
LIN {X 0,Y 286.477,Z 231.021,A -85,B 0,C 180,E1 -17345.83,E2 -17345.83} C_VEL
LIN {X 0,Y 284.244,Z 296.755,A -85,B 0,C 180,E1 -17347.898,E2 -17347.898} C_VEL
LIN {X 0,Y 283.392,Z 311.043,A -85,B 0,C 180,E1 -17348.64,E2 -17348.64} C_VEL
LIN {X 0,Y 282.292,Z 323.824,A -85,B 0,C 180,E1 -17349.603,E2 -17349.603} C_VEL
LIN {X 0,Y 281.085,Z 336.115,A -85,B 0,C 180,E1 -17350.844,E2 -17350.844} C_VEL
LIN {X 0,Y 279.813,Z 347.228,A -85,B 0,C 180,E1 -17352.271,E2 -17352.271} C_VEL
LIN {X 0,Y 278.627,Z 358.313,A -85,B 0,C 180,E1 -17354.081,E2 -17354.081} C_VEL
LIN {X 0,Y 277.453,Z 368.136,A -85,B 0,C 180,E1 -17356.077,E2 -17356.077} C_VEL
LIN {X 0,Y 276.435,Z 376.67,A -85,B 0,C 180,E1 -17358.266,E2 -17358.266} C_VEL
LIN {X 0,Y 275.863,Z 383.541,A -85,B 0,C 180,E1 -17360.469,E2 -17360.469} C_VEL
LIN {X 0,Y 275.503,Z 388.979,A -85,B 0,C 180,E1 -17362.673,E2 -17362.673} C_VEL
LIN {X 0,Y 275.333,Z 392.603,A -85,B 0,C 180,E1 -17364.559,E2 -17364.559} C_VEL
LIN {X 0,Y 275.329,Z 396.199,A -85,B 0,C 180,E1 -17367.075,E2 -17367.075} C_VEL
LIN {X 0,Y 275.271,Z 397.627,A -85,B 0,C 180,E1 -17368.538,E2 -17368.538} C_VEL
LIN {X 0,Y 275.279,Z 398.618,A -85,B 0,C 180,E1 -17370.001,E2 -17370.001} C_VEL
LIN {X 0,Y 275.255,Z 399.192,A -85,B 0,C 180,E1 -17371.464,E2 -17371.464} C_VEL
LIN {X 0,Y 275.243,Z 399.348,A -85,B 0,C 180,E1 -17372.928,E2 -17372.928} C_VEL
LIN {X 0,Y 275.245,Z 398.718,A -85,B 0,C 180,E1 -17375.247,E2 -17375.247} C_VEL
LIN {X 0,Y 275.518,Z 397.256,A -85,B 0,C 180,E1 -17377.329,E2 -17377.329} C_VEL
LIN {X 0,Y 275.859,Z 395.742,A -85,B 0,C 180,E1 -17378.794,E2 -17378.794} C_VEL
LIN {X 0,Y 276.598,Z 392.624,A -85,B 0,C 180,E1 -17380.987,E2 -17380.987} C_VEL
LIN {X 0,Y 277.663,Z 388.451,A -85,B 0,C 180,E1 -17383.169,E2 -17383.169} C_VEL
LIN {X 0,Y 279.243,Z 383.15,A -85,B 0,C 180,E1 -17385.324,E2 -17385.324} C_VEL
LIN {X 0,Y 281.166,Z 376.524,A -85,B 0,C 180,E1 -17387.456,E2 -17387.456} C_VEL
LIN {X 0,Y 283.313,Z 368.36,A -85,B 0,C 180,E1 -17389.566,E2 -17389.566} C_VEL
LIN {X 0,Y 285.516,Z 360.071,A -85,B 0,C 180,E1 -17391.29,E2 -17391.29} C_VEL
LIN {X 0,Y 288.045,Z 350.06,A -85,B 0,C 180,E1 -17392.98,E2 -17392.98} C_VEL
LIN {X 0,Y 290.588,Z 338.967,A -85,B 0,C 180,E1 -17394.469,E2 -17394.469} C_VEL
LIN {X 0,Y 293.011,Z 326.666,A -85,B 0,C 180,E1 -17395.77,E2 -17395.77} C_VEL
LIN {X 0,Y 294.836,Z 315.874,A -85,B 0,C 180,E1 -17396.644,E2 -17396.644} C_VEL
LIN {X 0,Y 296.75,Z 302.696,A -85,B 0,C 180,E1 -17397.41,E2 -17397.41} C_VEL
LIN {X 0,Y 297.885,Z 289.436,A -85,B 0,C 180,E1 -17397.965,E2 -17397.965} C_VEL
LIN {X 0,Y 301.283,Z 235.366,A -85,B 0,C 180,E1 -17399.7,E2 -17399.7} C_VEL
LIN {X 0,Y 299.463,Z 221.401,A -85,B 0,C 180,E1 -17400.635,E2 -17400.635} C_VEL
LIN {X 0,Y 298.369,Z 215.699,A -85,B 0,C 180,E1 -17401.092,E2 -17401.092} C_VEL
LIN {X 0,Y 292.986,Z 203.721,A -85,B 0,C 180,E1 -17402.701,E2 -17402.701} C_VEL
LIN {X 0,Y 288.245,Z 194.959,A -85,B 0,C 180,E1 -17404.161,E2 -17404.161} C_VEL
LIN {X 0,Y 284.89,Z 189.21,A -85,B 0,C 180,E1 -17405.275,E2 -17405.275} C_VEL
LIN {X 0,Y 282.226,Z 184.676,A -85,B 0,C 180,E1 -17406.199,E2 -17406.199} C_VEL
LIN {X 0,Y 280.578,Z 179.163,A -85,B 0,C 180,E1 -17409.059,E2 -17409.059} C_VEL
LIN {X 0,Y 278.991,Z 174.303,A -85,B 0,C 180,E1 -17412.002,E2 -17412.002} C_VEL
LIN {X 0,Y 277.196,Z 168.946,A -85,B 0,C 180,E1 -17415.885,E2 -17415.885} C_VEL
LIN {X 0,Y 277.2,Z 168.947,A -85,B 0,C 180,E1 -17419.519,E2 -17419.519} C_VEL
LIN {X 0,Y 277.255,Z 168.947,A -85,B 0,C 180,E1 -17422.529,E2 -17422.529} C_VEL
LIN {X 0,Y 277.249,Z 168.946,A -85,B 0,C 180,E1 -17426.105,E2 -17426.105} C_VEL
LIN {X 0,Y 277.266,Z 168.942,A -85,B 0,C 180,E1 -17429.539,E2 -17429.539} C_VEL
LIN {X 0,Y 277.292,Z 168.942,A -85,B 0,C 180,E1 -17432.857,E2 -17432.857} C_VEL
LIN {X 0,Y 277.264,Z 168.943,A -85,B 0,C 180,E1 -17436.074,E2 -17436.074} C_VEL
LIN {X 0,Y 277.283,Z 168.945,A -85,B 0,C 180,E1 -17440.762,E2 -17440.762} C_VEL
LIN {X 0,Y 277.386,Z 168.934,A -85,B 0,C 180,E1 -17445.323,E2 -17445.323} C_VEL
LIN {X 0,Y 277.398,Z 168.938,A -85,B 0,C 180,E1 -17446.073,E2 -17446.073} C_VEL
LIN {X 0,Y 279.233,Z 174.109,A -85,B 0,C 180,E1 -17449.853,E2 -17449.853} C_VEL
LIN {X 0,Y 280.152,Z 176.462,A -85,B 0,C 180,E1 -17451.278,E2 -17451.278} C_VEL
LIN {X 0,Y 282.764,Z 180.424,A -85,B 0,C 180,E1 -17452.232,E2 -17452.232} C_VEL
LIN {X 0,Y 284.32,Z 182.665,A -85,B 0,C 180,E1 -17452.753,E2 -17452.753} C_VEL
LIN {X 0,Y 290.395,Z 192.278,A -85,B 0,C 180,E1 -17454.714,E2 -17454.714} C_VEL
LIN {X 0,Y 293.306,Z 196.966,A -85,B 0,C 180,E1 -17455.565,E2 -17455.565} C_VEL
LIN {X 0,Y 298.022,Z 206.024,A -85,B 0,C 180,E1 -17456.935,E2 -17456.935} C_VEL
LIN {X 0,Y 302.311,Z 216.062,A -85,B 0,C 180,E1 -17458.158,E2 -17458.158} C_VEL
LIN {X 0,Y 301.961,Z 223.302,A -85,B 0,C 180,E1 -17458.416,E2 -17458.416} C_VEL
LIN {X 0,Y 297.839,Z 283.964,A -85,B 0,C 180,E1 -17460.381,E2 -17460.381} C_VEL
LIN {X 0,Y 296.342,Z 297.982,A -85,B 0,C 180,E1 -17461.104,E2 -17461.104} C_VEL
LIN {X 0,Y 294.506,Z 310.914,A -85,B 0,C 180,E1 -17462.077,E2 -17462.077} C_VEL
LIN {X 0,Y 292.301,Z 323.507,A -85,B 0,C 180,E1 -17463.345,E2 -17463.345} C_VEL
LIN {X 0,Y 289.932,Z 334.716,A -85,B 0,C 180,E1 -17464.801,E2 -17464.801} C_VEL
LIN {X 0,Y 287.414,Z 345.085,A -85,B 0,C 180,E1 -17466.494,E2 -17466.494} C_VEL
LIN {X 0,Y 285.153,Z 353.365,A -85,B 0,C 180,E1 -17468.148,E2 -17468.148} C_VEL
LIN {X 0,Y 283.089,Z 360.886,A -85,B 0,C 180,E1 -17470.008,E2 -17470.008} C_VEL
LIN {X 0,Y 281.159,Z 367.366,A -85,B 0,C 180,E1 -17471.987,E2 -17471.987} C_VEL
LIN {X 0,Y 279.606,Z 372.229,A -85,B 0,C 180,E1 -17473.815,E2 -17473.815} C_VEL
LIN {X 0,Y 278.072,Z 377.124,A -85,B 0,C 180,E1 -17476.172,E2 -17476.172} C_VEL
LIN {X 0,Y 276.938,Z 380.677,A -85,B 0,C 180,E1 -17478.495,E2 -17478.495} C_VEL
LIN {X 0,Y 276.07,Z 383.13,A -85,B 0,C 180,E1 -17480.88,E2 -17480.88} C_VEL
LIN {X 0,Y 275.448,Z 384.459,A -85,B 0,C 180,E1 -17483.285,E2 -17483.285} C_VEL
LIN {X 0,Y 275.088,Z 384.661,A -85,B 0,C 180,E1 -17485.743,E2 -17485.743} C_VEL
LIN {X 0,Y 274.953,Z 384.164,A -85,B 0,C 180,E1 -17487.394,E2 -17487.394} C_VEL
LIN {X 0,Y 274.969,Z 382.586,A -85,B 0,C 180,E1 -17489.654,E2 -17489.654} C_VEL
LIN {X 0,Y 275.252,Z 379.215,A -85,B 0,C 180,E1 -17492.425,E2 -17492.425} C_VEL
LIN {X 0,Y 275.608,Z 375.117,A -85,B 0,C 180,E1 -17494.735,E2 -17494.735} C_VEL
LIN {X 0,Y 276.095,Z 369.312,A -85,B 0,C 180,E1 -17497.198,E2 -17497.198} C_VEL
LIN {X 0,Y 276.822,Z 362.628,A -85,B 0,C 180,E1 -17499.399,E2 -17499.399} C_VEL
LIN {X 0,Y 277.754,Z 354.134,A -85,B 0,C 180,E1 -17501.622,E2 -17501.622} C_VEL
LIN {X 0,Y 278.722,Z 345.76,A -85,B 0,C 180,E1 -17503.403,E2 -17503.403} C_VEL
LIN {X 0,Y 279.786,Z 336.391,A -85,B 0,C 180,E1 -17505.043,E2 -17505.043} C_VEL
LIN {X 0,Y 280.929,Z 326.042,A -85,B 0,C 180,E1 -17506.511,E2 -17506.511} C_VEL
LIN {X 0,Y 282.192,Z 313.681,A -85,B 0,C 180,E1 -17507.901,E2 -17507.901} C_VEL
LIN {X 0,Y 283.151,Z 301.828,A -85,B 0,C 180,E1 -17508.933,E2 -17508.933} C_VEL
LIN {X 0,Y 283.993,Z 287.667,A -85,B 0,C 180,E1 -17509.819,E2 -17509.819} C_VEL
LIN {X 0,Y 284.672,Z 274.43,A -85,B 0,C 180,E1 -17510.351,E2 -17510.351} C_VEL
LIN {X 0,Y 286.938,Z 206.23,A -85,B 0,C 180,E1 -17512.462,E2 -17512.462} C_VEL
LIN {X 0,Y 284.893,Z 194.497,A -85,B 0,C 180,E1 -17512.98,E2 -17512.98} C_VEL
LIN {X 0,Y 278.195,Z 173.279,A -85,B 0,C 180,E1 -17514.165,E2 -17514.165} C_VEL
LIN {X 0,Y 277.331,Z 168.938,A -85,B 0,C 180,E1 -17515.786,E2 -17515.786} C_VEL
LIN {X 0,Y 277.233,Z 168.95,A -85,B 0,C 180,E1 -17519.534,E2 -17519.534} C_VEL
LIN {X 0,Y 277.255,Z 168.948,A -85,B 0,C 180,E1 -17522.852,E2 -17522.852} C_VEL
LIN {X 0,Y 277.26,Z 168.949,A -85,B 0,C 180,E1 -17526.072,E2 -17526.072} C_VEL
LIN {X 0,Y 277.281,Z 168.944,A -85,B 0,C 180,E1 -17530.76,E2 -17530.76} C_VEL
LIN {X 0,Y 277.375,Z 168.932,A -85,B 0,C 180,E1 -17535.321,E2 -17535.321} C_VEL
LIN {X 0,Y 277.458,Z 168.924,A -85,B 0,C 180,E1 -17539.786,E2 -17539.786} C_VEL
LIN {X 0,Y 277.604,Z 168.903,A -85,B 0,C 180,E1 -17542.727,E2 -17542.727} C_VEL
LIN {X 0,Y 277.808,Z 168.877,A -85,B 0,C 180,E1 -17548.549,E2 -17548.549} C_VEL
LIN {X 0,Y 277.808,Z 168.879,A -85,B 0,C 180,E1 -17551.448,E2 -17551.448} C_VEL
LIN {X 0,Y 277.602,Z 168.904,A -85,B 0,C 180,E1 -17557.271,E2 -17557.271} C_VEL
LIN {X 0,Y 277.456,Z 168.922,A -85,B 0,C 180,E1 -17560.212,E2 -17560.212} C_VEL
LIN {X 0,Y 277.372,Z 168.932,A -85,B 0,C 180,E1 -17564.676,E2 -17564.676} C_VEL
LIN {X 0,Y 277.276,Z 168.947,A -85,B 0,C 180,E1 -17569.237,E2 -17569.237} C_VEL
LIN {X 0,Y 277.255,Z 168.946,A -85,B 0,C 180,E1 -17573.926,E2 -17573.926} C_VEL
LIN {X 0,Y 277.266,Z 168.948,A -85,B 0,C 180,E1 -17577.48,E2 -17577.48} C_VEL
LIN {X 0,Y 277.247,Z 168.948,A -85,B 0,C 180,E1 -17580.471,E2 -17580.471} C_VEL
LIN {X 0,Y 277.244,Z 168.947,A -85,B 0,C 180,E1 -17583.894,E2 -17583.894} C_VEL
LIN {X 0,Y 277.253,Z 168.948,A -85,B 0,C 180,E1 -17587.47,E2 -17587.47} C_VEL
LIN {X 0,Y 277.181,Z 168.956,A -85,B 0,C 180,E1 -17591.24,E2 -17591.24} C_VEL
LIN {X 0,Y 277.17,Z 168.959,A -85,B 0,C 180,E1 -17595.231,E2 -17595.231} C_VEL
LIN {X 0,Y 277.18,Z 168.96,A -85,B 0,C 180,E1 -17598.757,E2 -17598.757} C_VEL
LIN {X 0,Y 277.251,Z 168.949,A -85,B 0,C 180,E1 -17602.527,E2 -17602.527} C_VEL
LIN {X 0,Y 277.241,Z 168.949,A -85,B 0,C 180,E1 -17606.103,E2 -17606.103} C_VEL
LIN {X 0,Y 277.257,Z 168.945,A -85,B 0,C 180,E1 -17609.537,E2 -17609.537} C_VEL
LIN {X 0,Y 277.283,Z 168.945,A -85,B 0,C 180,E1 -17612.856,E2 -17612.856} C_VEL
LIN {X 0,Y 277.249,Z 168.948,A -85,B 0,C 180,E1 -17616.072,E2 -17616.072} C_VEL
LIN {X 0,Y 277.272,Z 168.946,A -85,B 0,C 180,E1 -17620.76,E2 -17620.76} C_VEL
LIN {X 0,Y 277.364,Z 168.931,A -85,B 0,C 180,E1 -17625.322,E2 -17625.322} C_VEL
LIN {X 0,Y 277.394,Z 168.93,A -85,B 0,C 180,E1 -17628.737,E2 -17628.737} C_VEL
LIN {X 0,Y 276.751,Z 169.012,A -85,B 0,C 180,E1 -17629.951,E2 -17629.951} C_VEL
LIN {X 0,Y 273.948,Z 169.361,A -85,B 0,C 180,E1 -17631.93,E2 -17631.93} C_VEL
LIN {X 0,Y 271.544,Z 169.658,A -85,B 0,C 180,E1 -17633.537,E2 -17633.537} C_VEL
LIN {X 0,Y 270.487,Z 169.789,A -85,B 0,C 180,E1 -17634.782,E2 -17634.782} C_VEL
LIN {X 0,Y 270.387,Z 169.801,A -85,B 0,C 180,E1 -17635.203,E2 -17635.203} C_VEL
LIN {X 0,Y 270.762,Z 169.756,A -85,B 0,C 180,E1 -17638.512,E2 -17638.512} C_VEL
LIN {X 0,Y 270.762,Z 169.756,A -85,B 0,C 180,E1 -17641.487,E2 -17641.487} C_VEL
LIN {X 0,Y 270.555,Z 169.783,A -85,B 0,C 180,E1 -17647.462,E2 -17647.462} C_VEL
LIN {X 0,Y 270.378,Z 169.802,A -85,B 0,C 180,E1 -17650.483,E2 -17650.483} C_VEL
LIN {X 0,Y 270.331,Z 169.81,A -85,B 0,C 180,E1 -17655.068,E2 -17655.068} C_VEL
LIN {X 0,Y 270.211,Z 169.826,A -85,B 0,C 180,E1 -17659.762,E2 -17659.762} C_VEL
LIN {X 0,Y 270.175,Z 169.828,A -85,B 0,C 180,E1 -17664.436,E2 -17664.436} C_VEL
LIN {X 0,Y 270.189,Z 169.827,A -85,B 0,C 180,E1 -17667.918,E2 -17667.918} C_VEL
LIN {X 0,Y 270.167,Z 169.834,A -85,B 0,C 180,E1 -17671.35,E2 -17671.35} C_VEL
LIN {X 0,Y 270.191,Z 169.828,A -85,B 0,C 180,E1 -17674.907,E2 -17674.907} C_VEL
LIN {X 0,Y 270.192,Z 169.827,A -85,B 0,C 180,E1 -17678.711,E2 -17678.711} C_VEL
LIN {X 0,Y 270.142,Z 169.836,A -85,B 0,C 180,E1 -17683.246,E2 -17683.246} C_VEL
LIN {X 0,Y 270.146,Z 169.834,A -85,B 0,C 180,E1 -17687.439,E2 -17687.439} C_VEL
LIN {X 0,Y 270.203,Z 169.826,A -85,B 0,C 180,E1 -17691.375,E2 -17691.375} C_VEL
LIN {X 0,Y 270.194,Z 169.829,A -85,B 0,C 180,E1 -17695.095,E2 -17695.095} C_VEL
LIN {X 0,Y 270.23,Z 169.913,A -85,B 0,C 180,E1 -17697.397,E2 -17697.397} C_VEL
LIN {X 0,Y 272.46,Z 181.223,A -85,B 0,C 180,E1 -17701.285,E2 -17701.285} C_VEL
LIN {X 0,Y 273.785,Z 188.111,A -85,B 0,C 180,E1 -17703.567,E2 -17703.567} C_VEL
LIN {X 0,Y 275.08,Z 194.039,A -85,B 0,C 180,E1 -17703.862,E2 -17703.862} C_VEL
LIN {X 0,Y 279.619,Z 231.846,A -85,B 0,C 180,E1 -17705.462,E2 -17705.462} C_VEL
LIN {X 0,Y 277.352,Z 296.752,A -85,B 0,C 180,E1 -17707.564,E2 -17707.564} C_VEL
LIN {X 0,Y 276.495,Z 310.228,A -85,B 0,C 180,E1 -17708.276,E2 -17708.276} C_VEL
LIN {X 0,Y 275.397,Z 323.211,A -85,B 0,C 180,E1 -17709.264,E2 -17709.264} C_VEL
LIN {X 0,Y 274.156,Z 335.58,A -85,B 0,C 180,E1 -17710.535,E2 -17710.535} C_VEL
LIN {X 0,Y 272.85,Z 346.765,A -85,B 0,C 180,E1 -17711.997,E2 -17711.997} C_VEL
LIN {X 0,Y 271.663,Z 356.895,A -85,B 0,C 180,E1 -17713.661,E2 -17713.661} C_VEL
LIN {X 0,Y 270.653,Z 365.264,A -85,B 0,C 180,E1 -17715.336,E2 -17715.336} C_VEL
LIN {X 0,Y 269.617,Z 374.398,A -85,B 0,C 180,E1 -17717.583,E2 -17717.583} C_VEL
LIN {X 0,Y 268.914,Z 381.682,A -85,B 0,C 180,E1 -17719.841,E2 -17719.841} C_VEL
LIN {X 0,Y 268.458,Z 388.288,A -85,B 0,C 180,E1 -17722.48,E2 -17722.48} C_VEL
LIN {X 0,Y 268.261,Z 392.309,A -85,B 0,C 180,E1 -17724.586,E2 -17724.586} C_VEL
LIN {X 0,Y 268.235,Z 395.715,A -85,B 0,C 180,E1 -17726.998,E2 -17726.998} C_VEL
LIN {X 0,Y 268.199,Z 397.24,A -85,B 0,C 180,E1 -17728.5,E2 -17728.5} C_VEL
LIN {X 0,Y 268.203,Z 398.283,A -85,B 0,C 180,E1 -17730.001,E2 -17730.001} C_VEL
LIN {X 0,Y 268.181,Z 398.909,A -85,B 0,C 180,E1 -17731.503,E2 -17731.503} C_VEL
LIN {X 0,Y 268.155,Z 399.127,A -85,B 0,C 180,E1 -17733.006,E2 -17733.006} C_VEL
LIN {X 0,Y 268.155,Z 398.677,A -85,B 0,C 180,E1 -17735.171,E2 -17735.171} C_VEL
LIN {X 0,Y 268.476,Z 397.23,A -85,B 0,C 180,E1 -17737.522,E2 -17737.522} C_VEL
LIN {X 0,Y 268.832,Z 395.78,A -85,B 0,C 180,E1 -17739.026,E2 -17739.026} C_VEL
LIN {X 0,Y 269.629,Z 392.779,A -85,B 0,C 180,E1 -17741.275,E2 -17741.275} C_VEL
LIN {X 0,Y 270.74,Z 388.75,A -85,B 0,C 180,E1 -17743.512,E2 -17743.512} C_VEL
LIN {X 0,Y 272.435,Z 383.582,A -85,B 0,C 180,E1 -17745.717,E2 -17745.717} C_VEL
LIN {X 0,Y 274.434,Z 377.139,A -85,B 0,C 180,E1 -17747.898,E2 -17747.898} C_VEL
LIN {X 0,Y 276.701,Z 369.16,A -85,B 0,C 180,E1 -17750.054,E2 -17750.054} C_VEL
LIN {X 0,Y 279.434,Z 359.367,A -85,B 0,C 180,E1 -17752.165,E2 -17752.165} C_VEL
LIN {X 0,Y 282.189,Z 349.268,A -85,B 0,C 180,E1 -17753.874,E2 -17753.874} C_VEL
LIN {X 0,Y 284.884,Z 338.039,A -85,B 0,C 180,E1 -17755.382,E2 -17755.382} C_VEL
LIN {X 0,Y 287.408,Z 325.547,A -85,B 0,C 180,E1 -17756.702,E2 -17756.702} C_VEL
LIN {X 0,Y 289.574,Z 313.25,A -85,B 0,C 180,E1 -17757.657,E2 -17757.657} C_VEL
LIN {X 0,Y 291.517,Z 299.467,A -85,B 0,C 180,E1 -17758.435,E2 -17758.435} C_VEL
LIN {X 0,Y 292.825,Z 283.295,A -85,B 0,C 180,E1 -17759.038,E2 -17759.038} C_VEL
LIN {X 0,Y 295.922,Z 236.167,A -85,B 0,C 180,E1 -17760.599,E2 -17760.599} C_VEL
LIN {X 0,Y 294.185,Z 222.936,A -85,B 0,C 180,E1 -17761.53,E2 -17761.53} C_VEL
LIN {X 0,Y 293.41,Z 219.037,A -85,B 0,C 180,E1 -17761.866,E2 -17761.866} C_VEL
LIN {X 0,Y 288.822,Z 208.495,A -85,B 0,C 180,E1 -17763.34,E2 -17763.34} C_VEL
LIN {X 0,Y 284.547,Z 200.281,A -85,B 0,C 180,E1 -17764.745,E2 -17764.745} C_VEL
LIN {X 0,Y 281.102,Z 194.358,A -85,B 0,C 180,E1 -17765.932,E2 -17765.932} C_VEL
LIN {X 0,Y 278.023,Z 189.255,A -85,B 0,C 180,E1 -17767.068,E2 -17767.068} C_VEL
LIN {X 0,Y 274.916,Z 184.261,A -85,B 0,C 180,E1 -17768.293,E2 -17768.293} C_VEL
LIN {X 0,Y 273.097,Z 178.474,A -85,B 0,C 180,E1 -17771.729,E2 -17771.729} C_VEL
LIN {X 0,Y 271.283,Z 173.192,A -85,B 0,C 180,E1 -17775.615,E2 -17775.615} C_VEL
LIN {X 0,Y 270.157,Z 169.821,A -85,B 0,C 180,E1 -17778.795,E2 -17778.795} C_VEL
LIN {X 0,Y 270.195,Z 169.818,A -85,B 0,C 180,E1 -17781.372,E2 -17781.372} C_VEL
LIN {X 0,Y 270.201,Z 169.827,A -85,B 0,C 180,E1 -17785.095,E2 -17785.095} C_VEL
LIN {X 0,Y 270.188,Z 169.823,A -85,B 0,C 180,E1 -17789.137,E2 -17789.137} C_VEL
LIN {X 0,Y 270.203,Z 169.82,A -85,B 0,C 180,E1 -17792.173,E2 -17792.173} C_VEL
LIN {X 0,Y 270.188,Z 169.828,A -85,B 0,C 180,E1 -17795.564,E2 -17795.564} C_VEL
LIN {X 0,Y 270.224,Z 169.823,A -85,B 0,C 180,E1 -17800.239,E2 -17800.239} C_VEL
LIN {X 0,Y 270.31,Z 170.012,A -85,B 0,C 180,E1 -17803.382,E2 -17803.382} C_VEL
LIN {X 0,Y 272.327,Z 175.425,A -85,B 0,C 180,E1 -17808.085,E2 -17808.085} C_VEL
LIN {X 0,Y 272.858,Z 176.97,A -85,B 0,C 180,E1 -17809.097,E2 -17809.097} C_VEL
LIN {X 0,Y 276.532,Z 181.836,A -85,B 0,C 180,E1 -17810.574,E2 -17810.574} C_VEL
LIN {X 0,Y 280.895,Z 188.295,A -85,B 0,C 180,E1 -17812.204,E2 -17812.204} C_VEL
LIN {X 0,Y 288.627,Z 200.664,A -85,B 0,C 180,E1 -17814.755,E2 -17814.755} C_VEL
LIN {X 0,Y 293.805,Z 210.89,A -85,B 0,C 180,E1 -17816.351,E2 -17816.351} C_VEL
LIN {X 0,Y 296.971,Z 218.582,A -85,B 0,C 180,E1 -17817.318,E2 -17817.318} C_VEL
LIN {X 0,Y 292.337,Z 284.593,A -85,B 0,C 180,E1 -17819.527,E2 -17819.527} C_VEL
LIN {X 0,Y 290.744,Z 298.394,A -85,B 0,C 180,E1 -17820.259,E2 -17820.259} C_VEL
LIN {X 0,Y 288.76,Z 311.445,A -85,B 0,C 180,E1 -17821.268,E2 -17821.268} C_VEL
LIN {X 0,Y 286.671,Z 322.863,A -85,B 0,C 180,E1 -17822.424,E2 -17822.424} C_VEL
LIN {X 0,Y 284.173,Z 334.278,A -85,B 0,C 180,E1 -17823.9,E2 -17823.9} C_VEL
LIN {X 0,Y 281.671,Z 344.168,A -85,B 0,C 180,E1 -17825.512,E2 -17825.512} C_VEL
LIN {X 0,Y 279.179,Z 352.774,A -85,B 0,C 180,E1 -17827.231,E2 -17827.231} C_VEL
LIN {X 0,Y 276.979,Z 360.257,A -85,B 0,C 180,E1 -17829.088,E2 -17829.088} C_VEL
LIN {X 0,Y 274.541,Z 367.885,A -85,B 0,C 180,E1 -17831.443,E2 -17831.443} C_VEL
LIN {X 0,Y 272.823,Z 372.925,A -85,B 0,C 180,E1 -17833.406,E2 -17833.406} C_VEL
LIN {X 0,Y 271.288,Z 377.394,A -85,B 0,C 180,E1 -17835.634,E2 -17835.634} C_VEL
LIN {X 0,Y 269.972,Z 381.14,A -85,B 0,C 180,E1 -17838.204,E2 -17838.204} C_VEL
LIN {X 0,Y 269.265,Z 383.006,A -85,B 0,C 180,E1 -17840.008,E2 -17840.008} C_VEL
LIN {X 0,Y 268.799,Z 384.04,A -85,B 0,C 180,E1 -17841.472,E2 -17841.472} C_VEL
LIN {X 0,Y 268.318,Z 384.852,A -85,B 0,C 180,E1 -17843.542,E2 -17843.542} C_VEL
LIN {X 0,Y 268.101,Z 384.959,A -85,B 0,C 180,E1 -17844.799,E2 -17844.799} C_VEL
LIN {X 0,Y 267.885,Z 384.474,A -85,B 0,C 180,E1 -17846.873,E2 -17846.873} C_VEL
LIN {X 0,Y 267.821,Z 383.775,A -85,B 0,C 180,E1 -17848.187,E2 -17848.187} C_VEL
LIN {X 0,Y 267.886,Z 382.229,A -85,B 0,C 180,E1 -17850.029,E2 -17850.029} C_VEL
LIN {X 0,Y 268.137,Z 379.384,A -85,B 0,C 180,E1 -17852.326,E2 -17852.326} C_VEL
LIN {X 0,Y 268.42,Z 376.152,A -85,B 0,C 180,E1 -17854.259,E2 -17854.259} C_VEL
LIN {X 0,Y 268.906,Z 370.165,A -85,B 0,C 180,E1 -17856.951,E2 -17856.951} C_VEL
LIN {X 0,Y 269.655,Z 363.707,A -85,B 0,C 180,E1 -17859.2,E2 -17859.2} C_VEL
LIN {X 0,Y 270.5,Z 356.219,A -85,B 0,C 180,E1 -17861.296,E2 -17861.296} C_VEL
LIN {X 0,Y 271.515,Z 347.564,A -85,B 0,C 180,E1 -17863.255,E2 -17863.255} C_VEL
LIN {X 0,Y 272.68,Z 337.331,A -85,B 0,C 180,E1 -17865.136,E2 -17865.136} C_VEL
LIN {X 0,Y 273.904,Z 326.554,A -85,B 0,C 180,E1 -17866.725,E2 -17866.725} C_VEL
LIN {X 0,Y 275.221,Z 314.218,A -85,B 0,C 180,E1 -17868.153,E2 -17868.153} C_VEL
LIN {X 0,Y 276.235,Z 301.951,A -85,B 0,C 180,E1 -17869.252,E2 -17869.252} C_VEL
LIN {X 0,Y 277.052,Z 288.297,A -85,B 0,C 180,E1 -17870.133,E2 -17870.133} C_VEL
LIN {X 0,Y 277.748,Z 275.678,A -85,B 0,C 180,E1 -17870.667,E2 -17870.667} C_VEL
LIN {X 0,Y 280.097,Z 206.644,A -85,B 0,C 180,E1 -17872.866,E2 -17872.866} C_VEL
LIN {X 0,Y 278.342,Z 196.636,A -85,B 0,C 180,E1 -17873.322,E2 -17873.322} C_VEL
LIN {X 0,Y 271.005,Z 173.502,A -85,B 0,C 180,E1 -17874.644,E2 -17874.644} C_VEL
LIN {X 0,Y 270.281,Z 169.817,A -85,B 0,C 180,E1 -17876.008,E2 -17876.008} C_VEL
LIN {X 0,Y 270.161,Z 169.835,A -85,B 0,C 180,E1 -17880.377,E2 -17880.377} C_VEL
LIN {X 0,Y 270.182,Z 169.829,A -85,B 0,C 180,E1 -17883.754,E2 -17883.754} C_VEL
LIN {X 0,Y 270.186,Z 169.828,A -85,B 0,C 180,E1 -17887.033,E2 -17887.033} C_VEL
LIN {X 0,Y 270.224,Z 169.827,A -85,B 0,C 180,E1 -17890.237,E2 -17890.237} C_VEL
LIN {X 0,Y 270.343,Z 169.808,A -85,B 0,C 180,E1 -17894.931,E2 -17894.931} C_VEL
LIN {X 0,Y 270.39,Z 169.803,A -85,B 0,C 180,E1 -17899.516,E2 -17899.516} C_VEL
LIN {X 0,Y 270.566,Z 169.781,A -85,B 0,C 180,E1 -17902.536,E2 -17902.536} C_VEL
LIN {X 0,Y 270.773,Z 169.753,A -85,B 0,C 180,E1 -17908.511,E2 -17908.511} C_VEL
LIN {X 0,Y 270.773,Z 169.755,A -85,B 0,C 180,E1 -17911.486,E2 -17911.486} C_VEL
LIN {X 0,Y 270.564,Z 169.782,A -85,B 0,C 180,E1 -17917.461,E2 -17917.461} C_VEL
LIN {X 0,Y 270.388,Z 169.801,A -85,B 0,C 180,E1 -17920.482,E2 -17920.482} C_VEL
LIN {X 0,Y 270.34,Z 169.809,A -85,B 0,C 180,E1 -17925.067,E2 -17925.067} C_VEL
LIN {X 0,Y 270.219,Z 169.825,A -85,B 0,C 180,E1 -17929.76,E2 -17929.76} C_VEL
LIN {X 0,Y 270.182,Z 169.826,A -85,B 0,C 180,E1 -17934.434,E2 -17934.434} C_VEL
LIN {X 0,Y 270.196,Z 169.826,A -85,B 0,C 180,E1 -17937.916,E2 -17937.916} C_VEL
LIN {X 0,Y 270.173,Z 169.831,A -85,B 0,C 180,E1 -17941.348,E2 -17941.348} C_VEL
LIN {X 0,Y 270.196,Z 169.828,A -85,B 0,C 180,E1 -17944.905,E2 -17944.905} C_VEL
LIN {X 0,Y 270.196,Z 169.828,A -85,B 0,C 180,E1 -17948.709,E2 -17948.709} C_VEL
LIN {X 0,Y 270.145,Z 169.834,A -85,B 0,C 180,E1 -17953.244,E2 -17953.244} C_VEL
LIN {X 0,Y 270.148,Z 169.832,A -85,B 0,C 180,E1 -17957.436,E2 -17957.436} C_VEL
LIN {X 0,Y 270.204,Z 169.825,A -85,B 0,C 180,E1 -17961.373,E2 -17961.373} C_VEL
LIN {X 0,Y 270.194,Z 169.828,A -85,B 0,C 180,E1 -17965.093,E2 -17965.093} C_VEL
LIN {X 0,Y 270.179,Z 169.828,A -85,B 0,C 180,E1 -17969.135,E2 -17969.135} C_VEL
LIN {X 0,Y 270.194,Z 169.828,A -85,B 0,C 180,E1 -17972.171,E2 -17972.171} C_VEL
LIN {X 0,Y 270.176,Z 169.828,A -85,B 0,C 180,E1 -17975.563,E2 -17975.563} C_VEL
LIN {X 0,Y 270.214,Z 169.827,A -85,B 0,C 180,E1 -17980.237,E2 -17980.237} C_VEL
LIN {X 0,Y 270.332,Z 169.808,A -85,B 0,C 180,E1 -17984.931,E2 -17984.931} C_VEL
LIN {X 0,Y 270.379,Z 169.804,A -85,B 0,C 180,E1 -17989.516,E2 -17989.516} C_VEL
LIN {X 0,Y 270.555,Z 169.781,A -85,B 0,C 180,E1 -17992.537,E2 -17992.537} C_VEL
LIN {X 0,Y 270.387,Z 169.801,A -85,B 0,C 180,E1 -17995.203,E2 -17995.203} C_VEL
LIN {X 0,Y 269.753,Z 169.885,A -85,B 0,C 180,E1 -17996.449,E2 -17996.449} C_VEL
LIN {X 0,Y 267.147,Z 170.213,A -85,B 0,C 180,E1 -17998.487,E2 -17998.487} C_VEL
LIN {X 0,Y 264.071,Z 170.591,A -85,B 0,C 180,E1 -18000.988,E2 -18000.988} C_VEL
LIN {X 0,Y 263.664,Z 170.638,A -85,B 0,C 180,E1 -18001.849,E2 -18001.849} C_VEL
LIN {X 0,Y 263.519,Z 170.661,A -85,B 0,C 180,E1 -18007.663,E2 -18007.663} C_VEL
LIN {X 0,Y 263.322,Z 170.68,A -85,B 0,C 180,E1 -18010.767,E2 -18010.767} C_VEL
LIN {X 0,Y 263.28,Z 170.691,A -85,B 0,C 180,E1 -18015.482,E2 -18015.482} C_VEL
LIN {X 0,Y 263.199,Z 170.697,A -85,B 0,C 180,E1 -18020.312,E2 -18020.312} C_VEL
LIN {X 0,Y 263.119,Z 170.711,A -85,B 0,C 180,E1 -18025.3,E2 -18025.3} C_VEL
LIN {X 0,Y 263.125,Z 170.706,A -85,B 0,C 180,E1 -18028.736,E2 -18028.736} C_VEL
LIN {X 0,Y 263.122,Z 170.707,A -85,B 0,C 180,E1 -18032.29,E2 -18032.29} C_VEL
LIN {X 0,Y 263.169,Z 170.7,A -85,B 0,C 180,E1 -18036.762,E2 -18036.762} C_VEL
LIN {X 0,Y 263.085,Z 170.712,A -85,B 0,C 180,E1 -18039.876,E2 -18039.876} C_VEL
LIN {X 0,Y 263.07,Z 170.714,A -85,B 0,C 180,E1 -18043.995,E2 -18043.995} C_VEL
LIN {X 0,Y 263.075,Z 170.714,A -85,B 0,C 180,E1 -18048.419,E2 -18048.419} C_VEL
LIN {X 0,Y 263.152,Z 170.704,A -85,B 0,C 180,E1 -18052.104,E2 -18052.104} C_VEL
LIN {X 0,Y 263.147,Z 170.704,A -85,B 0,C 180,E1 -18055.887,E2 -18055.887} C_VEL
LIN {X 0,Y 263.198,Z 170.839,A -85,B 0,C 180,E1 -18057.098,E2 -18057.098} C_VEL
LIN {X 0,Y 265.338,Z 181.7,A -85,B 0,C 180,E1 -18060.935,E2 -18060.935} C_VEL
LIN {X 0,Y 266.548,Z 187.964,A -85,B 0,C 180,E1 -18063.064,E2 -18063.064} C_VEL
LIN {X 0,Y 268.364,Z 195.283,A -85,B 0,C 180,E1 -18063.455,E2 -18063.455} C_VEL
LIN {X 0,Y 272.783,Z 232.215,A -85,B 0,C 180,E1 -18065.059,E2 -18065.059} C_VEL
LIN {X 0,Y 270.459,Z 296.719,A -85,B 0,C 180,E1 -18067.212,E2 -18067.212} C_VEL
LIN {X 0,Y 269.554,Z 310.807,A -85,B 0,C 180,E1 -18067.99,E2 -18067.99} C_VEL
LIN {X 0,Y 268.516,Z 322.529,A -85,B 0,C 180,E1 -18068.908,E2 -18068.908} C_VEL
LIN {X 0,Y 267.24,Z 334.969,A -85,B 0,C 180,E1 -18070.21,E2 -18070.21} C_VEL
LIN {X 0,Y 265.917,Z 346.105,A -85,B 0,C 180,E1 -18071.694,E2 -18071.694} C_VEL
LIN {X 0,Y 264.645,Z 356.405,A -85,B 0,C 180,E1 -18073.414,E2 -18073.414} C_VEL
LIN {X 0,Y 263.56,Z 365.658,A -85,B 0,C 180,E1 -18075.327,E2 -18075.327} C_VEL
LIN {X 0,Y 262.466,Z 374.67,A -85,B 0,C 180,E1 -18077.632,E2 -18077.632} C_VEL
LIN {X 0,Y 261.777,Z 381.832,A -85,B 0,C 180,E1 -18079.951,E2 -18079.951} C_VEL
LIN {X 0,Y 261.385,Z 387.529,A -85,B 0,C 180,E1 -18082.275,E2 -18082.275} C_VEL
LIN {X 0,Y 261.165,Z 392.065,A -85,B 0,C 180,E1 -18084.67,E2 -18084.67} C_VEL
LIN {X 0,Y 261.145,Z 395.21,A -85,B 0,C 180,E1 -18086.916,E2 -18086.916} C_VEL
LIN {X 0,Y 261.128,Z 396.806,A -85,B 0,C 180,E1 -18088.459,E2 -18088.459} C_VEL
LIN {X 0,Y 261.129,Z 397.947,A -85,B 0,C 180,E1 -18090.001,E2 -18090.001} C_VEL
LIN {X 0,Y 261.108,Z 398.626,A -85,B 0,C 180,E1 -18091.544,E2 -18091.544} C_VEL
LIN {X 0,Y 261.069,Z 398.896,A -85,B 0,C 180,E1 -18093.088,E2 -18093.088} C_VEL
LIN {X 0,Y 261.049,Z 398.646,A -85,B 0,C 180,E1 -18095.05,E2 -18095.05} C_VEL
LIN {X 0,Y 261.41,Z 397.221,A -85,B 0,C 180,E1 -18097.727,E2 -18097.727} C_VEL
LIN {X 0,Y 261.795,Z 395.837,A -85,B 0,C 180,E1 -18099.27,E2 -18099.27} C_VEL
LIN {X 0,Y 262.653,Z 392.954,A -85,B 0,C 180,E1 -18101.578,E2 -18101.578} C_VEL
LIN {X 0,Y 263.829,Z 389.045,A -85,B 0,C 180,E1 -18103.873,E2 -18103.873} C_VEL
LIN {X 0,Y 265.642,Z 384.001,A -85,B 0,C 180,E1 -18106.13,E2 -18106.13} C_VEL
LIN {X 0,Y 267.722,Z 377.757,A -85,B 0,C 180,E1 -18108.363,E2 -18108.363} C_VEL
LIN {X 0,Y 270.109,Z 370.068,A -85,B 0,C 180,E1 -18110.565,E2 -18110.565} C_VEL
LIN {X 0,Y 272.967,Z 360.491,A -85,B 0,C 180,E1 -18112.72,E2 -18112.72} C_VEL
LIN {X 0,Y 276.133,Z 349.611,A -85,B 0,C 180,E1 -18114.632,E2 -18114.632} C_VEL
LIN {X 0,Y 279.273,Z 337.195,A -85,B 0,C 180,E1 -18116.331,E2 -18116.331} C_VEL
LIN {X 0,Y 281.914,Z 324.64,A -85,B 0,C 180,E1 -18117.667,E2 -18117.667} C_VEL
LIN {X 0,Y 284.439,Z 311.098,A -85,B 0,C 180,E1 -18118.704,E2 -18118.704} C_VEL
LIN {X 0,Y 286.256,Z 298.116,A -85,B 0,C 180,E1 -18119.409,E2 -18119.409} C_VEL
LIN {X 0,Y 287.835,Z 278.01,A -85,B 0,C 180,E1 -18120.141,E2 -18120.141} C_VEL
LIN {X 0,Y 290.684,Z 237.446,A -85,B 0,C 180,E1 -18121.514,E2 -18121.514} C_VEL
LIN {X 0,Y 288.89,Z 223.121,A -85,B 0,C 180,E1 -18122.584,E2 -18122.584} C_VEL
LIN {X 0,Y 284.604,Z 213.063,A -85,B 0,C 180,E1 -18124.033,E2 -18124.033} C_VEL
LIN {X 0,Y 280.44,Z 204.805,A -85,B 0,C 180,E1 -18125.504,E2 -18125.504} C_VEL
LIN {X 0,Y 277.389,Z 199.457,A -85,B 0,C 180,E1 -18126.615,E2 -18126.615} C_VEL
LIN {X 0,Y 274.638,Z 194.716,A -85,B 0,C 180,E1 -18127.7,E2 -18127.7} C_VEL
LIN {X 0,Y 271.142,Z 189.196,A -85,B 0,C 180,E1 -18129.153,E2 -18129.153} C_VEL
LIN {X 0,Y 267.859,Z 184.372,A -85,B 0,C 180,E1 -18130.646,E2 -18130.646} C_VEL
LIN {X 0,Y 267.43,Z 183.473,A -85,B 0,C 180,E1 -18130.915,E2 -18130.915} C_VEL
LIN {X 0,Y 265.819,Z 178.55,A -85,B 0,C 180,E1 -18134.451,E2 -18134.451} C_VEL
LIN {X 0,Y 264.304,Z 174.231,A -85,B 0,C 180,E1 -18138.336,E2 -18138.336} C_VEL
LIN {X 0,Y 263.151,Z 170.704,A -85,B 0,C 180,E1 -18142.896,E2 -18142.896} C_VEL
LIN {X 0,Y 263.155,Z 170.702,A -85,B 0,C 180,E1 -18145.886,E2 -18145.886} C_VEL
LIN {X 0,Y 263.129,Z 170.702,A -85,B 0,C 180,E1 -18149.504,E2 -18149.504} C_VEL
LIN {X 0,Y 263.131,Z 170.707,A -85,B 0,C 180,E1 -18152.996,E2 -18152.996} C_VEL
LIN {X 0,Y 263.121,Z 170.703,A -85,B 0,C 180,E1 -18156.381,E2 -18156.381} C_VEL
LIN {X 0,Y 263.181,Z 170.729,A -85,B 0,C 180,E1 -18159.173,E2 -18159.173} C_VEL
LIN {X 0,Y 264.377,Z 173.791,A -85,B 0,C 180,E1 -18163.14,E2 -18163.14} C_VEL
LIN {X 0,Y 265.716,Z 177.505,A -85,B 0,C 180,E1 -18166.536,E2 -18166.536} C_VEL
LIN {X 0,Y 268.93,Z 181.842,A -85,B 0,C 180,E1 -18168.097,E2 -18168.097} C_VEL
LIN {X 0,Y 270.584,Z 183.985,A -85,B 0,C 180,E1 -18168.834,E2 -18168.834} C_VEL
LIN {X 0,Y 274.297,Z 188.958,A -85,B 0,C 180,E1 -18170.367,E2 -18170.367} C_VEL
LIN {X 0,Y 277.741,Z 194.224,A -85,B 0,C 180,E1 -18171.703,E2 -18171.703} C_VEL
LIN {X 0,Y 284.72,Z 205.738,A -85,B 0,C 180,E1 -18174.134,E2 -18174.134} C_VEL
LIN {X 0,Y 289.706,Z 215.873,A -85,B 0,C 180,E1 -18175.755,E2 -18175.755} C_VEL
LIN {X 0,Y 291.799,Z 221.334,A -85,B 0,C 180,E1 -18176.457,E2 -18176.457} C_VEL
LIN {X 0,Y 286.992,Z 284.591,A -85,B 0,C 180,E1 -18178.597,E2 -18178.597} C_VEL
LIN {X 0,Y 285.401,Z 297.808,A -85,B 0,C 180,E1 -18179.295,E2 -18179.295} C_VEL
LIN {X 0,Y 283.67,Z 309.332,A -85,B 0,C 180,E1 -18180.162,E2 -18180.162} C_VEL
LIN {X 0,Y 281.482,Z 320.881,A -85,B 0,C 180,E1 -18181.3,E2 -18181.3} C_VEL
LIN {X 0,Y 278.96,Z 331.954,A -85,B 0,C 180,E1 -18182.69,E2 -18182.69} C_VEL
LIN {X 0,Y 276.113,Z 342.707,A -85,B 0,C 180,E1 -18184.38,E2 -18184.38} C_VEL
LIN {X 0,Y 273.317,Z 352.23,A -85,B 0,C 180,E1 -18186.274,E2 -18186.274} C_VEL
LIN {X 0,Y 270.985,Z 359.609,A -85,B 0,C 180,E1 -18188.091,E2 -18188.091} C_VEL
LIN {X 0,Y 268.662,Z 366.465,A -85,B 0,C 180,E1 -18190.171,E2 -18190.171} C_VEL
LIN {X 0,Y 266.41,Z 372.683,A -85,B 0,C 180,E1 -18192.554,E2 -18192.554} C_VEL
LIN {X 0,Y 264.837,Z 376.841,A -85,B 0,C 180,E1 -18194.602,E2 -18194.602} C_VEL
LIN {X 0,Y 263.396,Z 380.644,A -85,B 0,C 180,E1 -18197.068,E2 -18197.068} C_VEL
LIN {X 0,Y 262.641,Z 382.501,A -85,B 0,C 180,E1 -18198.73,E2 -18198.73} C_VEL
LIN {X 0,Y 262.031,Z 383.87,A -85,B 0,C 180,E1 -18200.407,E2 -18200.407} C_VEL
LIN {X 0,Y 261.518,Z 384.773,A -85,B 0,C 180,E1 -18202.101,E2 -18202.101} C_VEL
LIN {X 0,Y 261.179,Z 385.133,A -85,B 0,C 180,E1 -18203.806,E2 -18203.806} C_VEL
LIN {X 0,Y 260.899,Z 385.027,A -85,B 0,C 180,E1 -18205.532,E2 -18205.532} C_VEL
LIN {X 0,Y 260.752,Z 384.372,A -85,B 0,C 180,E1 -18207.271,E2 -18207.271} C_VEL
LIN {X 0,Y 260.727,Z 383.176,A -85,B 0,C 180,E1 -18209.026,E2 -18209.026} C_VEL
LIN {X 0,Y 260.942,Z 380.317,A -85,B 0,C 180,E1 -18211.682,E2 -18211.682} C_VEL
LIN {X 0,Y 261.336,Z 375.949,A -85,B 0,C 180,E1 -18214.385,E2 -18214.385} C_VEL
LIN {X 0,Y 261.877,Z 369.853,A -85,B 0,C 180,E1 -18217.145,E2 -18217.145} C_VEL
LIN {X 0,Y 262.62,Z 363.302,A -85,B 0,C 180,E1 -18219.439,E2 -18219.439} C_VEL
LIN {X 0,Y 263.597,Z 354.783,A -85,B 0,C 180,E1 -18221.802,E2 -18221.802} C_VEL
LIN {X 0,Y 264.771,Z 345.064,A -85,B 0,C 180,E1 -18223.963,E2 -18223.963} C_VEL
LIN {X 0,Y 265.959,Z 334.868,A -85,B 0,C 180,E1 -18225.773,E2 -18225.773} C_VEL
LIN {X 0,Y 267.31,Z 323.406,A -85,B 0,C 180,E1 -18227.406,E2 -18227.406} C_VEL
LIN {X 0,Y 268.617,Z 310.985,A -85,B 0,C 180,E1 -18228.783,E2 -18228.783} C_VEL
LIN {X 0,Y 269.596,Z 298.591,A -85,B 0,C 180,E1 -18229.831,E2 -18229.831} C_VEL
LIN {X 0,Y 270.337,Z 285.614,A -85,B 0,C 180,E1 -18230.626,E2 -18230.626} C_VEL
LIN {X 0,Y 271.126,Z 267.646,A -85,B 0,C 180,E1 -18231.298,E2 -18231.298} C_VEL
LIN {X 0,Y 273.376,Z 208.08,A -85,B 0,C 180,E1 -18233.247,E2 -18233.247} C_VEL
LIN {X 0,Y 271.74,Z 198.684,A -85,B 0,C 180,E1 -18233.687,E2 -18233.687} C_VEL
LIN {X 0,Y 263.823,Z 173.681,A -85,B 0,C 180,E1 -18235.15,E2 -18235.15} C_VEL
LIN {X 0,Y 263.204,Z 170.699,A -85,B 0,C 180,E1 -18236.353,E2 -18236.353} C_VEL
LIN {X 0,Y 263.114,Z 170.709,A -85,B 0,C 180,E1 -18239.501,E2 -18239.501} C_VEL
LIN {X 0,Y 263.117,Z 170.709,A -85,B 0,C 180,E1 -18242.993,E2 -18242.993} C_VEL
LIN {X 0,Y 263.12,Z 170.711,A -85,B 0,C 180,E1 -18246.38,E2 -18246.38} C_VEL
LIN {X 0,Y 263.212,Z 170.697,A -85,B 0,C 180,E1 -18249.688,E2 -18249.688} C_VEL
LIN {X 0,Y 263.293,Z 170.688,A -85,B 0,C 180,E1 -18254.517,E2 -18254.517} C_VEL
LIN {X 0,Y 263.334,Z 170.681,A -85,B 0,C 180,E1 -18259.231,E2 -18259.231} C_VEL
LIN {X 0,Y 263.53,Z 170.658,A -85,B 0,C 180,E1 -18262.336,E2 -18262.336} C_VEL
LIN {X 0,Y 263.737,Z 170.63,A -85,B 0,C 180,E1 -18268.472,E2 -18268.472} C_VEL
LIN {X 0,Y 263.737,Z 170.632,A -85,B 0,C 180,E1 -18271.526,E2 -18271.526} C_VEL
LIN {X 0,Y 263.528,Z 170.659,A -85,B 0,C 180,E1 -18277.662,E2 -18277.662} C_VEL
LIN {X 0,Y 263.332,Z 170.681,A -85,B 0,C 180,E1 -18280.766,E2 -18280.766} C_VEL
LIN {X 0,Y 263.289,Z 170.689,A -85,B 0,C 180,E1 -18285.48,E2 -18285.48} C_VEL
LIN {X 0,Y 263.207,Z 170.696,A -85,B 0,C 180,E1 -18290.31,E2 -18290.31} C_VEL
LIN {X 0,Y 263.126,Z 170.709,A -85,B 0,C 180,E1 -18295.298,E2 -18295.298} C_VEL
LIN {X 0,Y 263.132,Z 170.707,A -85,B 0,C 180,E1 -18298.734,E2 -18298.734} C_VEL
LIN {X 0,Y 263.127,Z 170.706,A -85,B 0,C 180,E1 -18302.287,E2 -18302.287} C_VEL
LIN {X 0,Y 263.174,Z 170.703,A -85,B 0,C 180,E1 -18306.76,E2 -18306.76} C_VEL
LIN {X 0,Y 263.089,Z 170.711,A -85,B 0,C 180,E1 -18309.874,E2 -18309.874} C_VEL
LIN {X 0,Y 263.073,Z 170.713,A -85,B 0,C 180,E1 -18313.992,E2 -18313.992} C_VEL
LIN {X 0,Y 263.077,Z 170.714,A -85,B 0,C 180,E1 -18318.416,E2 -18318.416} C_VEL
LIN {X 0,Y 263.153,Z 170.703,A -85,B 0,C 180,E1 -18322.101,E2 -18322.101} C_VEL
LIN {X 0,Y 263.147,Z 170.704,A -85,B 0,C 180,E1 -18325.884,E2 -18325.884} C_VEL
LIN {X 0,Y 263.121,Z 170.706,A -85,B 0,C 180,E1 -18329.502,E2 -18329.502} C_VEL
LIN {X 0,Y 263.121,Z 170.708,A -85,B 0,C 180,E1 -18332.994,E2 -18332.994} C_VEL
LIN {X 0,Y 263.11,Z 170.711,A -85,B 0,C 180,E1 -18336.379,E2 -18336.379} C_VEL
LIN {X 0,Y 263.201,Z 170.697,A -85,B 0,C 180,E1 -18339.688,E2 -18339.688} C_VEL
LIN {X 0,Y 263.281,Z 170.688,A -85,B 0,C 180,E1 -18344.517,E2 -18344.517} C_VEL
LIN {X 0,Y 263.323,Z 170.682,A -85,B 0,C 180,E1 -18349.232,E2 -18349.232} C_VEL
LIN {X 0,Y 263.519,Z 170.659,A -85,B 0,C 180,E1 -18352.336,E2 -18352.336} C_VEL
LIN {X 0,Y 263.726,Z 170.633,A -85,B 0,C 180,E1 -18358.473,E2 -18358.473} C_VEL
LIN {X 0,Y 263.664,Z 170.638,A -85,B 0,C 180,E1 -18361.849,E2 -18361.849} C_VEL
LIN {X 0,Y 262.842,Z 170.742,A -85,B 0,C 180,E1 -18363.122,E2 -18363.122} C_VEL
LIN {X 0,Y 259.927,Z 171.105,A -85,B 0,C 180,E1 -18365.198,E2 -18365.198} C_VEL
LIN {X 0,Y 257.536,Z 171.404,A -85,B 0,C 180,E1 -18366.887,E2 -18366.887} C_VEL
LIN {X 0,Y 256.504,Z 171.533,A -85,B 0,C 180,E1 -18368.196,E2 -18368.196} C_VEL
LIN {X 0,Y 256.411,Z 171.542,A -85,B 0,C 180,E1 -18368.639,E2 -18368.639} C_VEL
LIN {X 0,Y 256.227,Z 171.565,A -85,B 0,C 180,E1 -18372.675,E2 -18372.675} C_VEL
LIN {X 0,Y 256.195,Z 171.57,A -85,B 0,C 180,E1 -18376.24,E2 -18376.24} C_VEL
LIN {X 0,Y 256.111,Z 171.581,A -85,B 0,C 180,E1 -18381.097,E2 -18381.097} C_VEL
LIN {X 0,Y 256.078,Z 171.586,A -85,B 0,C 180,E1 -18385.089,E2 -18385.089} C_VEL
LIN {X 0,Y 256.082,Z 171.583,A -85,B 0,C 180,E1 -18388.575,E2 -18388.575} C_VEL
LIN {X 0,Y 256.067,Z 171.587,A -85,B 0,C 180,E1 -18391.702,E2 -18391.702} C_VEL
LIN {X 0,Y 256.073,Z 171.587,A -85,B 0,C 180,E1 -18395.194,E2 -18395.194} C_VEL
LIN {X 0,Y 256.104,Z 171.584,A -85,B 0,C 180,E1 -18397.27,E2 -18397.27} C_VEL
LIN {X 0,Y 256.012,Z 171.596,A -85,B 0,C 180,E1 -18401.212,E2 -18401.212} C_VEL
LIN {X 0,Y 256.012,Z 171.594,A -85,B 0,C 180,E1 -18405.541,E2 -18405.541} C_VEL
LIN {X 0,Y 256.013,Z 171.597,A -85,B 0,C 180,E1 -18408.791,E2 -18408.791} C_VEL
LIN {X 0,Y 256.121,Z 171.583,A -85,B 0,C 180,E1 -18412.868,E2 -18412.868} C_VEL
LIN {X 0,Y 256.145,Z 171.679,A -85,B 0,C 180,E1 -18416.77,E2 -18416.77} C_VEL
LIN {X 0,Y 258.521,Z 183.777,A -85,B 0,C 180,E1 -18421.15,E2 -18421.15} C_VEL
LIN {X 0,Y 259.299,Z 187.774,A -85,B 0,C 180,E1 -18422.546,E2 -18422.546} C_VEL
LIN {X 0,Y 261.559,Z 195.716,A -85,B 0,C 180,E1 -18423.005,E2 -18423.005} C_VEL
LIN {X 0,Y 265.911,Z 233.167,A -85,B 0,C 180,E1 -18424.674,E2 -18424.674} C_VEL
LIN {X 0,Y 263.584,Z 296.068,A -85,B 0,C 180,E1 -18426.843,E2 -18426.843} C_VEL
LIN {X 0,Y 262.7,Z 309.553,A -85,B 0,C 180,E1 -18427.592,E2 -18427.592} C_VEL
LIN {X 0,Y 261.657,Z 321.543,A -85,B 0,C 180,E1 -18428.535,E2 -18428.535} C_VEL
LIN {X 0,Y 260.497,Z 332.6,A -85,B 0,C 180,E1 -18429.676,E2 -18429.676} C_VEL
LIN {X 0,Y 259.142,Z 344.232,A -85,B 0,C 180,E1 -18431.215,E2 -18431.215} C_VEL
LIN {X 0,Y 257.735,Z 354.772,A -85,B 0,C 180,E1 -18432.956,E2 -18432.956} C_VEL
LIN {X 0,Y 256.837,Z 362.551,A -85,B 0,C 180,E1 -18434.528,E2 -18434.528} C_VEL
LIN {X 0,Y 255.861,Z 370.707,A -85,B 0,C 180,E1 -18436.5,E2 -18436.5} C_VEL
LIN {X 0,Y 254.98,Z 378.631,A -85,B 0,C 180,E1 -18438.877,E2 -18438.877} C_VEL
LIN {X 0,Y 254.449,Z 384.96,A -85,B 0,C 180,E1 -18441.264,E2 -18441.264} C_VEL
LIN {X 0,Y 254.159,Z 389.933,A -85,B 0,C 180,E1 -18443.651,E2 -18443.651} C_VEL
LIN {X 0,Y 254.028,Z 393.695,A -85,B 0,C 180,E1 -18446.035,E2 -18446.035} C_VEL
LIN {X 0,Y 254.058,Z 396.36,A -85,B 0,C 180,E1 -18448.416,E2 -18448.416} C_VEL
LIN {X 0,Y 254.056,Z 397.58,A -85,B 0,C 180,E1 -18450.001,E2 -18450.001} C_VEL
LIN {X 0,Y 254.036,Z 398.339,A -85,B 0,C 180,E1 -18451.587,E2 -18451.587} C_VEL
LIN {X 0,Y 253.966,Z 398.662,A -85,B 0,C 180,E1 -18453.174,E2 -18453.174} C_VEL
LIN {X 0,Y 253.952,Z 398.56,A -85,B 0,C 180,E1 -18454.942,E2 -18454.942} C_VEL
LIN {X 0,Y 254.359,Z 397.221,A -85,B 0,C 180,E1 -18457.942,E2 -18457.942} C_VEL
LIN {X 0,Y 254.778,Z 395.895,A -85,B 0,C 180,E1 -18459.528,E2 -18459.528} C_VEL
LIN {X 0,Y 255.696,Z 393.129,A -85,B 0,C 180,E1 -18461.898,E2 -18461.898} C_VEL
LIN {X 0,Y 256.935,Z 389.374,A -85,B 0,C 180,E1 -18464.253,E2 -18464.253} C_VEL
LIN {X 0,Y 258.862,Z 384.508,A -85,B 0,C 180,E1 -18466.564,E2 -18466.564} C_VEL
LIN {X 0,Y 261.371,Z 377.404,A -85,B 0,C 180,E1 -18469.188,E2 -18469.188} C_VEL
LIN {X 0,Y 264.016,Z 369.508,A -85,B 0,C 180,E1 -18471.471,E2 -18471.471} C_VEL
LIN {X 0,Y 267.096,Z 359.898,A -85,B 0,C 180,E1 -18473.659,E2 -18473.659} C_VEL
LIN {X 0,Y 270.128,Z 350.105,A -85,B 0,C 180,E1 -18475.424,E2 -18475.424} C_VEL
LIN {X 0,Y 273.071,Z 339.294,A -85,B 0,C 180,E1 -18476.977,E2 -18476.977} C_VEL
LIN {X 0,Y 275.835,Z 327.321,A -85,B 0,C 180,E1 -18478.331,E2 -18478.331} C_VEL
LIN {X 0,Y 278.379,Z 314.819,A -85,B 0,C 180,E1 -18479.389,E2 -18479.389} C_VEL
LIN {X 0,Y 280.691,Z 300.24,A -85,B 0,C 180,E1 -18480.259,E2 -18480.259} C_VEL
LIN {X 0,Y 282.05,Z 286.524,A -85,B 0,C 180,E1 -18480.823,E2 -18480.823} C_VEL
LIN {X 0,Y 285.612,Z 238.813,A -85,B 0,C 180,E1 -18482.475,E2 -18482.475} C_VEL
LIN {X 0,Y 284.086,Z 226.343,A -85,B 0,C 180,E1 -18483.444,E2 -18483.444} C_VEL
LIN {X 0,Y 280.306,Z 217.185,A -85,B 0,C 180,E1 -18484.833,E2 -18484.833} C_VEL
LIN {X 0,Y 276.14,Z 208.946,A -85,B 0,C 180,E1 -18486.377,E2 -18486.377} C_VEL
LIN {X 0,Y 273.236,Z 203.628,A -85,B 0,C 180,E1 -18487.543,E2 -18487.543} C_VEL
LIN {X 0,Y 271.164,Z 200,A -85,B 0,C 180,E1 -18488.401,E2 -18488.401} C_VEL
LIN {X 0,Y 268.055,Z 194.913,A -85,B 0,C 180,E1 -18489.788,E2 -18489.788} C_VEL
LIN {X 0,Y 264.783,Z 189.804,A -85,B 0,C 180,E1 -18491.371,E2 -18491.371} C_VEL
LIN {X 0,Y 260.293,Z 183.525,A -85,B 0,C 180,E1 -18493.829,E2 -18493.829} C_VEL
LIN {X 0,Y 259.926,Z 182.7,A -85,B 0,C 180,E1 -18494.233,E2 -18494.233} C_VEL
LIN {X 0,Y 258.776,Z 179.345,A -85,B 0,C 180,E1 -18497.237,E2 -18497.237} C_VEL
LIN {X 0,Y 257.551,Z 175.987,A -85,B 0,C 180,E1 -18501.126,E2 -18501.126} C_VEL
LIN {X 0,Y 257.264,Z 174.635,A -85,B 0,C 180,E1 -18503.059,E2 -18503.059} C_VEL
LIN {X 0,Y 256.345,Z 172.766,A -85,B 0,C 180,E1 -18508.203,E2 -18508.203} C_VEL
LIN {X 0,Y 256.297,Z 172.528,A -85,B 0,C 180,E1 -18512.215,E2 -18512.215} C_VEL
LIN {X 0,Y 256.529,Z 173.346,A -85,B 0,C 180,E1 -18515.736,E2 -18515.736} C_VEL
LIN {X 0,Y 257.384,Z 174.864,A -85,B 0,C 180,E1 -18519.209,E2 -18519.209} C_VEL
LIN {X 0,Y 258.63,Z 178.134,A -85,B 0,C 180,E1 -18523.35,E2 -18523.35} C_VEL
LIN {X 0,Y 261.826,Z 182.423,A -85,B 0,C 180,E1 -18525.306,E2 -18525.306} C_VEL
LIN {X 0,Y 263.43,Z 184.163,A -85,B 0,C 180,E1 -18526.153,E2 -18526.153} C_VEL
LIN {X 0,Y 267.884,Z 190.141,A -85,B 0,C 180,E1 -18528.342,E2 -18528.342} C_VEL
LIN {X 0,Y 271.448,Z 195.202,A -85,B 0,C 180,E1 -18529.909,E2 -18529.909} C_VEL
LIN {X 0,Y 274.587,Z 200.09,A -85,B 0,C 180,E1 -18531.166,E2 -18531.166} C_VEL
LIN {X 0,Y 281.224,Z 211.485,A -85,B 0,C 180,E1 -18533.61,E2 -18533.61} C_VEL
LIN {X 0,Y 285.956,Z 221.562,A -85,B 0,C 180,E1 -18535.252,E2 -18535.252} C_VEL
LIN {X 0,Y 286.652,Z 223.411,A -85,B 0,C 180,E1 -18535.495,E2 -18535.495} C_VEL
LIN {X 0,Y 281.781,Z 284.564,A -85,B 0,C 180,E1 -18537.62,E2 -18537.62} C_VEL
LIN {X 0,Y 280.03,Z 298.253,A -85,B 0,C 180,E1 -18538.357,E2 -18538.357} C_VEL
LIN {X 0,Y 278.113,Z 310.166,A -85,B 0,C 180,E1 -18539.276,E2 -18539.276} C_VEL
LIN {X 0,Y 275.824,Z 321.616,A -85,B 0,C 180,E1 -18540.434,E2 -18540.434} C_VEL
LIN {X 0,Y 273.182,Z 332.621,A -85,B 0,C 180,E1 -18541.843,E2 -18541.843} C_VEL
LIN {X 0,Y 270.202,Z 343.182,A -85,B 0,C 180,E1 -18543.542,E2 -18543.542} C_VEL
LIN {X 0,Y 267.375,Z 352.182,A -85,B 0,C 180,E1 -18545.371,E2 -18545.371} C_VEL
LIN {X 0,Y 264.83,Z 359.663,A -85,B 0,C 180,E1 -18547.242,E2 -18547.242} C_VEL
LIN {X 0,Y 262.067,Z 367.389,A -85,B 0,C 180,E1 -18549.649,E2 -18549.649} C_VEL
LIN {X 0,Y 260.05,Z 372.564,A -85,B 0,C 180,E1 -18551.695,E2 -18551.695} C_VEL
LIN {X 0,Y 258.019,Z 377.511,A -85,B 0,C 180,E1 -18554.191,E2 -18554.191} C_VEL
LIN {X 0,Y 256.574,Z 380.912,A -85,B 0,C 180,E1 -18556.518,E2 -18556.518} C_VEL
LIN {X 0,Y 255.344,Z 383.659,A -85,B 0,C 180,E1 -18559.286,E2 -18559.286} C_VEL
LIN {X 0,Y 254.716,Z 384.707,A -85,B 0,C 180,E1 -18561.02,E2 -18561.02} C_VEL
LIN {X 0,Y 254.019,Z 385.389,A -85,B 0,C 180,E1 -18564.071,E2 -18564.071} C_VEL
LIN {X 0,Y 253.724,Z 384.885,A -85,B 0,C 180,E1 -18566.308,E2 -18566.308} C_VEL
LIN {X 0,Y 253.616,Z 383.904,A -85,B 0,C 180,E1 -18568.106,E2 -18568.106} C_VEL
LIN {X 0,Y 253.741,Z 381.346,A -85,B 0,C 180,E1 -18570.835,E2 -18570.835} C_VEL
LIN {X 0,Y 254.129,Z 377.427,A -85,B 0,C 180,E1 -18573.581,E2 -18573.581} C_VEL
LIN {X 0,Y 254.545,Z 372.377,A -85,B 0,C 180,E1 -18576.158,E2 -18576.158} C_VEL
LIN {X 0,Y 255.275,Z 365.614,A -85,B 0,C 180,E1 -18578.781,E2 -18578.781} C_VEL
LIN {X 0,Y 256.207,Z 357.798,A -85,B 0,C 180,E1 -18581.174,E2 -18581.174} C_VEL
LIN {X 0,Y 257.288,Z 349.004,A -85,B 0,C 180,E1 -18583.339,E2 -18583.339} C_VEL
LIN {X 0,Y 258.435,Z 339.264,A -85,B 0,C 180,E1 -18585.273,E2 -18585.273} C_VEL
LIN {X 0,Y 259.682,Z 328.859,A -85,B 0,C 180,E1 -18586.948,E2 -18586.948} C_VEL
LIN {X 0,Y 261.052,Z 316.846,A -85,B 0,C 180,E1 -18588.482,E2 -18588.482} C_VEL
LIN {X 0,Y 262.223,Z 304.281,A -85,B 0,C 180,E1 -18589.717,E2 -18589.717} C_VEL
LIN {X 0,Y 263.143,Z 290.736,A -85,B 0,C 180,E1 -18590.697,E2 -18590.697} C_VEL
LIN {X 0,Y 263.9,Z 276.759,A -85,B 0,C 180,E1 -18591.357,E2 -18591.357} C_VEL
LIN {X 0,Y 266.494,Z 208.53,A -85,B 0,C 180,E1 -18593.672,E2 -18593.672} C_VEL
LIN {X 0,Y 265.069,Z 200.507,A -85,B 0,C 180,E1 -18594.06,E2 -18594.06} C_VEL
LIN {X 0,Y 256.606,Z 173.842,A -85,B 0,C 180,E1 -18595.699,E2 -18595.699} C_VEL
LIN {X 0,Y 256.167,Z 171.576,A -85,B 0,C 180,E1 -18596.609,E2 -18596.609} C_VEL
LIN {X 0,Y 256.081,Z 171.585,A -85,B 0,C 180,E1 -18601.43,E2 -18601.43} C_VEL
LIN {X 0,Y 256.09,Z 171.584,A -85,B 0,C 180,E1 -18605.69,E2 -18605.69} C_VEL
LIN {X 0,Y 256.126,Z 171.579,A -85,B 0,C 180,E1 -18609.1,E2 -18609.1} C_VEL
LIN {X 0,Y 256.217,Z 171.572,A -85,B 0,C 180,E1 -18614.078,E2 -18614.078} C_VEL
LIN {X 0,Y 256.278,Z 171.56,A -85,B 0,C 180,E1 -18618.931,E2 -18618.931} C_VEL
LIN {X 0,Y 256.494,Z 171.536,A -85,B 0,C 180,E1 -18622.124,E2 -18622.124} C_VEL
LIN {X 0,Y 256.454,Z 171.538,A -85,B 0,C 180,E1 -18626.857,E2 -18626.857} C_VEL
LIN {X 0,Y 256.699,Z 171.507,A -85,B 0,C 180,E1 -18628.43,E2 -18628.43} C_VEL
LIN {X 0,Y 256.699,Z 171.508,A -85,B 0,C 180,E1 -18631.568,E2 -18631.568} C_VEL
LIN {X 0,Y 256.456,Z 171.537,A -85,B 0,C 180,E1 -18636.292,E2 -18636.292} C_VEL
LIN {X 0,Y 256.404,Z 171.545,A -85,B 0,C 180,E1 -18639.464,E2 -18639.464} C_VEL
LIN {X 0,Y 256.203,Z 171.569,A -85,B 0,C 180,E1 -18644.292,E2 -18644.292} C_VEL
LIN {X 0,Y 256.147,Z 171.579,A -85,B 0,C 180,E1 -18647.565,E2 -18647.565} C_VEL
LIN {X 0,Y 256.119,Z 171.582,A -85,B 0,C 180,E1 -18651.095,E2 -18651.095} C_VEL
LIN {X 0,Y 256.085,Z 171.585,A -85,B 0,C 180,E1 -18655.087,E2 -18655.087} C_VEL
LIN {X 0,Y 256.089,Z 171.584,A -85,B 0,C 180,E1 -18658.573,E2 -18658.573} C_VEL
LIN {X 0,Y 256.073,Z 171.585,A -85,B 0,C 180,E1 -18661.7,E2 -18661.7} C_VEL
LIN {X 0,Y 256.078,Z 171.588,A -85,B 0,C 180,E1 -18665.192,E2 -18665.192} C_VEL
LIN {X 0,Y 256.108,Z 171.583,A -85,B 0,C 180,E1 -18667.268,E2 -18667.268} C_VEL
LIN {X 0,Y 256.016,Z 171.592,A -85,B 0,C 180,E1 -18671.209,E2 -18671.209} C_VEL
LIN {X 0,Y 256.014,Z 171.593,A -85,B 0,C 180,E1 -18675.538,E2 -18675.538} C_VEL
LIN {X 0,Y 256.015,Z 171.595,A -85,B 0,C 180,E1 -18678.788,E2 -18678.788} C_VEL
LIN {X 0,Y 256.122,Z 171.582,A -85,B 0,C 180,E1 -18682.865,E2 -18682.865} C_VEL
LIN {X 0,Y 256.062,Z 171.589,A -85,B 0,C 180,E1 -18686.706,E2 -18686.706} C_VEL
LIN {X 0,Y 256.049,Z 171.59,A -85,B 0,C 180,E1 -18690.392,E2 -18690.392} C_VEL
LIN {X 0,Y 256.068,Z 171.587,A -85,B 0,C 180,E1 -18693.951,E2 -18693.951} C_VEL
LIN {X 0,Y 256.051,Z 171.586,A -85,B 0,C 180,E1 -18697.401,E2 -18697.401} C_VEL
LIN {X 0,Y 256.101,Z 171.583,A -85,B 0,C 180,E1 -18700.773,E2 -18700.773} C_VEL
LIN {X 0,Y 256.207,Z 171.571,A -85,B 0,C 180,E1 -18704.079,E2 -18704.079} C_VEL
LIN {X 0,Y 256.267,Z 171.561,A -85,B 0,C 180,E1 -18708.932,E2 -18708.932} C_VEL
LIN {X 0,Y 256.483,Z 171.537,A -85,B 0,C 180,E1 -18712.125,E2 -18712.125} C_VEL
LIN {X 0,Y 256.443,Z 171.539,A -85,B 0,C 180,E1 -18716.858,E2 -18716.858} C_VEL
LIN {X 0,Y 256.688,Z 171.51,A -85,B 0,C 180,E1 -18718.431,E2 -18718.431} C_VEL
LIN {X 0,Y 256.644,Z 171.513,A -85,B 0,C 180,E1 -18721.779,E2 -18721.779} C_VEL
LIN {X 0,Y 256.447,Z 171.54,A -85,B 0,C 180,E1 -18726.293,E2 -18726.293} C_VEL
LIN {X 0,Y 256.411,Z 171.542,A -85,B 0,C 180,E1 -18728.639,E2 -18728.639} C_VEL
LIN {X 0,Y 255.693,Z 171.633,A -85,B 0,C 180,E1 -18729.949,E2 -18729.949} C_VEL
LIN {X 0,Y 252.735,Z 172.002,A -85,B 0,C 180,E1 -18732.081,E2 -18732.081} C_VEL
LIN {X 0,Y 250.248,Z 172.314,A -85,B 0,C 180,E1 -18733.816,E2 -18733.816} C_VEL
LIN {X 0,Y 249.197,Z 172.443,A -85,B 0,C 180,E1 -18735.165,E2 -18735.165} C_VEL
LIN {X 0,Y 249.119,Z 172.448,A -85,B 0,C 180,E1 -18735.622,E2 -18735.622} C_VEL
LIN {X 0,Y 249.034,Z 172.463,A -85,B 0,C 180,E1 -18739.795,E2 -18739.795} C_VEL
LIN {X 0,Y 248.998,Z 172.469,A -85,B 0,C 180,E1 -18743.275,E2 -18743.275} C_VEL
LIN {X 0,Y 249.014,Z 172.464,A -85,B 0,C 180,E1 -18746.844,E2 -18746.844} C_VEL
LIN {X 0,Y 248.995,Z 172.467,A -85,B 0,C 180,E1 -18750.534,E2 -18750.534} C_VEL
LIN {X 0,Y 249.037,Z 172.464,A -85,B 0,C 180,E1 -18755.078,E2 -18755.078} C_VEL
LIN {X 0,Y 249.016,Z 172.464,A -85,B 0,C 180,E1 -18758.382,E2 -18758.382} C_VEL
LIN {X 0,Y 248.964,Z 172.472,A -85,B 0,C 180,E1 -18762.784,E2 -18762.784} C_VEL
LIN {X 0,Y 248.974,Z 172.472,A -85,B 0,C 180,E1 -18767.356,E2 -18767.356} C_VEL
LIN {X 0,Y 249.036,Z 172.463,A -85,B 0,C 180,E1 -18772.203,E2 -18772.203} C_VEL
LIN {X 0,Y 249.068,Z 172.548,A -85,B 0,C 180,E1 -18776.438,E2 -18776.438} C_VEL
LIN {X 0,Y 251.058,Z 182.621,A -85,B 0,C 180,E1 -18780.204,E2 -18780.204} C_VEL
LIN {X 0,Y 252.11,Z 187.74,A -85,B 0,C 180,E1 -18782.014,E2 -18782.014} C_VEL
LIN {X 0,Y 254.944,Z 197.812,A -85,B 0,C 180,E1 -18782.617,E2 -18782.617} C_VEL
LIN {X 0,Y 259.064,Z 233.971,A -85,B 0,C 180,E1 -18784.276,E2 -18784.276} C_VEL
LIN {X 0,Y 256.674,Z 296.416,A -85,B 0,C 180,E1 -18786.502,E2 -18786.502} C_VEL
LIN {X 0,Y 255.772,Z 309.72,A -85,B 0,C 180,E1 -18787.271,E2 -18787.271} C_VEL
LIN {X 0,Y 254.547,Z 322.608,A -85,B 0,C 180,E1 -18788.33,E2 -18788.33} C_VEL
LIN {X 0,Y 253.267,Z 334.968,A -85,B 0,C 180,E1 -18789.706,E2 -18789.706} C_VEL
LIN {X 0,Y 251.859,Z 346.145,A -85,B 0,C 180,E1 -18791.285,E2 -18791.285} C_VEL
LIN {X 0,Y 250.639,Z 355.382,A -85,B 0,C 180,E1 -18792.904,E2 -18792.904} C_VEL
LIN {X 0,Y 249.523,Z 364.652,A -85,B 0,C 180,E1 -18794.9,E2 -18794.9} C_VEL
LIN {X 0,Y 248.362,Z 373.781,A -85,B 0,C 180,E1 -18797.333,E2 -18797.333} C_VEL
LIN {X 0,Y 247.628,Z 381.071,A -85,B 0,C 180,E1 -18799.784,E2 -18799.784} C_VEL
LIN {X 0,Y 247.27,Z 385.99,A -85,B 0,C 180,E1 -18801.831,E2 -18801.831} C_VEL
LIN {X 0,Y 247.021,Z 391.374,A -85,B 0,C 180,E1 -18804.737,E2 -18804.737} C_VEL
LIN {X 0,Y 246.973,Z 394.173,A -85,B 0,C 180,E1 -18806.739,E2 -18806.739} C_VEL
LIN {X 0,Y 246.988,Z 395.885,A -85,B 0,C 180,E1 -18808.371,E2 -18808.371} C_VEL
LIN {X 0,Y 246.985,Z 397.164,A -85,B 0,C 180,E1 -18810.001,E2 -18810.001} C_VEL
LIN {X 0,Y 246.964,Z 398.023,A -85,B 0,C 180,E1 -18811.632,E2 -18811.632} C_VEL
LIN {X 0,Y 246.868,Z 398.427,A -85,B 0,C 180,E1 -18813.265,E2 -18813.265} C_VEL
LIN {X 0,Y 246.882,Z 398.412,A -85,B 0,C 180,E1 -18814.9,E2 -18814.9} C_VEL
LIN {X 0,Y 247.307,Z 397.194,A -85,B 0,C 180,E1 -18818.17,E2 -18818.17} C_VEL
LIN {X 0,Y 247.777,Z 395.964,A -85,B 0,C 180,E1 -18819.8,E2 -18819.8} C_VEL
LIN {X 0,Y 248.732,Z 393.348,A -85,B 0,C 180,E1 -18822.236,E2 -18822.236} C_VEL
LIN {X 0,Y 250.057,Z 389.728,A -85,B 0,C 180,E1 -18824.654,E2 -18824.654} C_VEL
LIN {X 0,Y 252.099,Z 385.009,A -85,B 0,C 180,E1 -18827.022,E2 -18827.022} C_VEL
LIN {X 0,Y 254.361,Z 379.088,A -85,B 0,C 180,E1 -18829.365,E2 -18829.365} C_VEL
LIN {X 0,Y 256.876,Z 372.096,A -85,B 0,C 180,E1 -18831.593,E2 -18831.593} C_VEL
LIN {X 0,Y 260.143,Z 362.874,A -85,B 0,C 180,E1 -18833.907,E2 -18833.907} C_VEL
LIN {X 0,Y 263.533,Z 352.728,A -85,B 0,C 180,E1 -18835.895,E2 -18835.895} C_VEL
LIN {X 0,Y 266.923,Z 341.268,A -85,B 0,C 180,E1 -18837.651,E2 -18837.651} C_VEL
LIN {X 0,Y 269.816,Z 330.018,A -85,B 0,C 180,E1 -18839.022,E2 -18839.022} C_VEL
LIN {X 0,Y 272.161,Z 319.468,A -85,B 0,C 180,E1 -18840.023,E2 -18840.023} C_VEL
LIN {X 0,Y 274.564,Z 306.903,A -85,B 0,C 180,E1 -18840.901,E2 -18840.901} C_VEL
LIN {X 0,Y 276.326,Z 293.626,A -85,B 0,C 180,E1 -18841.587,E2 -18841.587} C_VEL
LIN {X 0,Y 280.66,Z 240.366,A -85,B 0,C 180,E1 -18843.458,E2 -18843.458} C_VEL
LIN {X 0,Y 279.501,Z 229.766,A -85,B 0,C 180,E1 -18844.317,E2 -18844.317} C_VEL
LIN {X 0,Y 275.426,Z 219.799,A -85,B 0,C 180,E1 -18845.913,E2 -18845.913} C_VEL
LIN {X 0,Y 270.541,Z 210.194,A -85,B 0,C 180,E1 -18847.922,E2 -18847.922} C_VEL
LIN {X 0,Y 267.755,Z 205.28,A -85,B 0,C 180,E1 -18849.138,E2 -18849.138} C_VEL
LIN {X 0,Y 265.067,Z 200.7,A -85,B 0,C 180,E1 -18850.418,E2 -18850.418} C_VEL
LIN {X 0,Y 261.343,Z 194.84,A -85,B 0,C 180,E1 -18852.353,E2 -18852.353} C_VEL
LIN {X 0,Y 257.221,Z 188.802,A -85,B 0,C 180,E1 -18854.825,E2 -18854.825} C_VEL
LIN {X 0,Y 252.421,Z 182.062,A -85,B 0,C 180,E1 -18858.627,E2 -18858.627} C_VEL
LIN {X 0,Y 251.59,Z 179.402,A -85,B 0,C 180,E1 -18862.081,E2 -18862.081} C_VEL
LIN {X 0,Y 251.118,Z 178.212,A -85,B 0,C 180,E1 -18864.256,E2 -18864.256} C_VEL
LIN {X 0,Y 250.604,Z 177.032,A -85,B 0,C 180,E1 -18867.803,E2 -18867.803} C_VEL
LIN {X 0,Y 250.528,Z 176.67,A -85,B 0,C 180,E1 -18871.517,E2 -18871.517} C_VEL
LIN {X 0,Y 250.728,Z 177.306,A -85,B 0,C 180,E1 -18875.137,E2 -18875.137} C_VEL
LIN {X 0,Y 251.576,Z 178.933,A -85,B 0,C 180,E1 -18878.92,E2 -18878.92} C_VEL
